//Reset
	IF x_Reset THEN
		x_Speicher:=FALSE;
	END_IF
	
//Ausgang schreiben
	x_Aus:=x_Speicher;

END_FUNCTION_BLOCK

// Converters/Converter2Punkt
(*Der Eingang f_Ein wird anhand des Bereiches von f_Ein_Min f_Ein_Max auf den Bereich f_Aus_Min und f_Aus_Max berechnet und auf den Ausgang f_Aus gegeben.
*)
FUNCTION_BLOCK Converter2Punkt
(*
Versionsverlauf: 
Version		|Autor	|Bemerkung
------------------------------------------------------------------------------------------------------------ 
17.06.00	|ShgB	|erste Freigabe 
17.06.01	|ShgB	|von Integer auf Real geändert 
17.08.00	|LeaF	|Freigabe	

*)
VAR_INPUT
	f_Ein:REAL;//Eingang
	f_Ein_Min:REAL;//Eingangsbereich Minimum
	f_Ein_Max:REAL;//Eingangsbereich Maximum
	f_Aus_Min:REAL;//Ausgangsbereich Minimum
	f_Aus_Max:REAL;//Ausgangsbereich Maximum
END_VAR
VAR_OUTPUT
	f_Aus:REAL;//Ausgang
END_VAR
VAR
END_VAR

IF f_Ein_Max-f_Ein_Min <> 0 THEN
	f_Aus:=(f_Aus_Max-f_Aus_Min)/(f_Ein_Max-f_Ein_Min)*(f_Ein-f_Ein_Min)+f_Aus_Min;
ELSE
	f_Aus:=f_Aus_Max;
END_IF

END_FUNCTION_BLOCK

// Math/Maximum
(*Gibt den grössten der angeschlossenen Werten aus.
*)
FUNCTION_BLOCK Maximum
(*
Versionsverlauf: 
Version		|Autor	|Bemerkung
------------------------------------------------------------------------------------------------------------ 
17.06.00	|Shgb	|erste Freigabe 
17.06.01	|ShgB	|von Integer auf Real geändert	 
17.08.00	|LeaF	|Freigabe

*)
VAR_INPUT
	f_Ein1 :REAL:=0.00001;//Wert 1
	f_Ein2 :REAL:=0.00001;//Wert 2
	f_Ein3 :REAL:=0.00001;//Wert 3
	f_Ein4 :REAL:=0.00001;//Wert 4
	f_Ein5 :REAL:=0.00001;//Wert 5
	f_Ein6 :REAL:=0.00001;//Wert 6
	f_Ein7 :REAL:=0.00001;//Wert 7
	f_Ein8 :REAL:=0.00001;//Wert 8
END_VAR
VAR_OUTPUT
	f_Aus:REAL;//Grösste Wert
END_VAR
VAR
	i_Arraypos:INT;
	af_Array: ARRAY [1..8] OF REAL;
END_VAR

// Werte in Array platzieren
	af_Array[1]:=f_Ein1;
	af_Array[2]:=f_Ein2;
	af_Array[3]:=f_Ein3;
	af_Array[4]:=f_Ein4;
	af_Array[5]:=f_Ein5;
	af_Array[6]:=f_Ein6;
	af_Array[7]:=f_Ein7;
	af_Array[8]:=f_Ein8;
	
//Zahlen die kleiner als 0 sind
	f_Aus := af_Array[1];	
	
//Auswertung der grössten Zahl
	FOR i_Arraypos:=2 TO 8 DO
		IF af_Array[i_Arraypos] >= f_Aus AND af_Array[i_Arraypos] <> 0.00001 THEN
			f_Aus := af_Array[i_Arraypos];
		END_IF
	END_FOR

END_FUNCTION_BLOCK

// Converters/Int_to_Druck
(*Der analoge Wert der Eingangskarte wird von einem 16 bit Integer in einen REAL Wert umgewandelt und ein Offset dazu addiert.
Standardmässig ist der Eingangsbereich von 0 - 32767 eingestellt. Sollte dieser nicht übereinstimmen kann der Bereich angepasst werden.
*)
FUNCTION_BLOCK Int_to_Druck
(*
Versionsverlauf: 
Version		|Autor	|Bemerkung
------------------------------------------------------------------------------------------------------------ 
17.06.00	|Shgb	|erste Freigabe  
17.08.00	|LeaF	|Freigabe

*)
VAR_INPUT
	i_Ein:INT;//Digitaler Eingangswert
END_VAR
VAR_INPUT PERSISTENT
	i_Ein_Min:INT:=0;//Eingangsbereich Minimum
	i_Ein_Max:INT:=32767;//Eingangsbereich Maximum
	f_Aus_Min:REAL;//Minimum des Drucktransmitters
	f_Aus_Max:REAL;//Maximum des Drucktransmitters
	f_Offset:REAL;//Offset der dazu addiert wird
END_VAR
VAR_OUTPUT
	f_Aus:REAL;//Druck im REAL Format
END_VAR
VAR//GUI Variablen
	f_GUI_Input:REAL;
END_VAR

IF i_Ein_Max-i_Ein_Min <> 0 THEN
	f_Aus:=(f_Aus_Max-f_Aus_Min)/(i_Ein_Max-i_Ein_Min)*(i_Ein-i_Ein_Min)+f_Aus_Min+f_Offset;
ELSE
	f_Aus:=f_Aus_Min;
END_IF

f_GUI_Input:=f_Aus-f_Offset;

END_FUNCTION_BLOCK

// Converters/Int_to_Temperature
(*Wandelt die Temperatur im INT Format, die von der Eingangskarte kommt, in eine Temperatur in REAL Format um und rechnet einen Offset dazu.
*)
FUNCTION_BLOCK Int_to_Temperature
(*
Versionsverlauf: 
Version		|Autor	|Bemerkung
------------------------------------------------------------------------------------------------------------ 
17.06.00	|Shgb	|erste Freigabe  
17.08.00	|LeaF	|Freigabe

*)
VAR_INPUT
	i_Ein:INT;//Temperatur von Karte
END_VAR
VAR_INPUT PERSISTENT
	f_Offset:REAL;//Offset der dazu addiert wird
END_VAR
VAR_OUTPUT
	f_Temperatur:REAL;//Ausgang REAL
END_VAR
VAR//GUI Variablen
	f_GUI_Input:REAL;
END_VAR

f_Temperatur:=i_Ein/10.0+f_Offset;
f_GUI_Input:=i_Ein/10.0;

END_FUNCTION_BLOCK

// Converters/Prozent_to_Int
(*Wandelt eine Prozentangabe vom Format REAL in eine Integer Zahl für die analoge Augangskarte um.
Standardmässig ist der Eingangsbereich von 0 - 32767 eingestellt. Sollte dieser nicht übereinstimmen kann der Bereich angepasst werden.
*)
FUNCTION_BLOCK Prozent_to_Int
(*
Versionsverlauf: 
Version		|Autor	|Bemerkung
------------------------------------------------------------------------------------------------------------ 
17.06.00	|Shgb	|erste Freigabe 
17.08.00	|LeaF	|Freigabe 

*)
VAR_INPUT
	f_Ein:REAL;//Eingang in Prozent
END_VAR
VAR_INPUT PERSISTENT
	i_Aus_Min:INT:=0;//Eingangsbereich Minimum
	i_Aus_Max:INT:=32767;//eingangsbereich Maximum
END_VAR
VAR_OUTPUT
	f_Aus:INT;//Ausgang
END_VAR
VAR
END_VAR

f_Aus:=real_to_int((i_Aus_Max-i_Aus_Min)*f_Ein/100.0);

END_FUNCTION_BLOCK

// Converters/Time_to_Timestruct
(*Wandelt die Eingangsvariable vom Typ TIME in ein TIMESTRUCT um.
*)
FUNCTION_BLOCK Time_to_Timestruct
(*
Versionsverlauf: 
Version		|Autor	|Bemerkung
------------------------------------------------------------------------------------------------------------ 
17.06.00	|Shgb	|erste Freigabe 	 
17.08.00	|LeaF	|Freigabe

*)
VAR_INPUT
	t_Ein:TIME;//Eingang
END_VAR
VAR_OUTPUT
	t_Aus:timestruct;//Ausgang
END_VAR
VAR
	OT:OTSTRUCT;
END_VAR

OT:=TIME_TO_OTSTRUCT(t_Ein);
t_Aus.wMilliseconds:=ot.wMilliseconds;
t_Aus.wSecond:=ot.wSecond;
t_Aus.wMinute:=ot.wMinute;
t_Aus.wHour:=ot.wHour;
t_Aus.wDay:=ot.wDay+ot.wWeek*7;

END_FUNCTION_BLOCK

// Converters/Timestruct_to_Time
(*Wandelt einen TIMESTRUCT in die Ausgangsvariable vom Typ TIME um.
*)
FUNCTION_BLOCK Timestruct_to_Time
(*
Versionsverlauf: 
Version		|Autor	|Bemerkung
------------------------------------------------------------------------------------------------------------ 
17.06.00	|Shgb	|erste Freigabe  
17.08.00	|LeaF	|Freigabe	

*)
VAR_INPUT
	t_Ein:timestruct;//Eingang
END_VAR
VAR_OUTPUT
	t_Aus:TIME;//Ausgang
END_VAR
VAR
END_VAR

t_Aus:=DINT_TO_TIME(t_Ein.wMilliseconds
					+ t_Ein.wSecond*1000
					+ t_Ein.wMinute*1000*60
					+ t_Ein.wHour*1000*60*60
					+ t_Ein.wDay*1000*60*60*24);

END_FUNCTION_BLOCK

// Druck_Temp/R1234ze
(*Wandelt den Druck in die Entsprechende Temperatur um. Die Druck-Temperatur Werte sind in der Nassdampftabelle in den Globalen Variablen hinterlegt.
*)
FUNCTION_BLOCK R1234ze
(*
Versionsverlauf: 
Version		|Autor	|Bemerkung
------------------------------------------------------------------------------------------------------------ 
17.06.00	|Shgb	|erste Freigabe 
17.06.01	|ShgB	|von Integer auf Real geändert	 
17.08.00	|LeaF	|Freigabe

*)
VAR_INPUT
	f_ND:REAL;//Druck für Verdampfungstemperatur
	f_HD:REAL;//Druck für Kondensationstemperatur
END_VAR
VAR_OUTPUT
	f_VerdTemp:REAL;//Verdampfungstemperatur
	f_KondTemp:REAL;//Kondensationstemperatur
END_VAR
VAR
END_VAR

//Niederdruck
	f_VerdTemp:=Nassdampftabelle.R1234ze[REAL_TO_INT(f_ND*100)+100]/10.0;
	
//Hochdruck
	f_KondTemp:=Nassdampftabelle.R1234ze[REAL_TO_INT(f_HD*100)+100]/10.0;

END_FUNCTION_BLOCK

// Druck_Temp/R134a
(*Wandelt den Druck in die Entsprechende Temperatur um. Die Druck-Temperatur Werte sind in der Nassdampftabelle in den Globalen Variablen hinterlegt.
*)
FUNCTION_BLOCK R134a
(*
Versionsverlauf: 
Version		|Autor	|Bemerkung
------------------------------------------------------------------------------------------------------------ 
17.06.00	|Shgb	|erste Freigabe 
17.06.01	|ShgB	|von Integer auf Real geändert	 
17.08.00	|LeaF	|Freigabe

*)
VAR_INPUT
	f_ND:REAL;//Druck für Verdampfungstemperatur
	f_HD:REAL;//Druck für Kondensationstemperatur
END_VAR
VAR_OUTPUT
	f_VerdTemp:REAL;//Verdampfungstemperatur
	f_KondTemp:REAL;//Kondensationstemperatur
END_VAR
VAR
END_VAR

//Niederdruck
	f_VerdTemp:=Nassdampftabelle.R134a[REAL_TO_INT(f_ND*100)+100]/10.0;
	
//Hochdruck
	f_KondTemp:=Nassdampftabelle.R134a[REAL_TO_INT(f_HD*100)+100]/10.0;

END_FUNCTION_BLOCK

// Druck_Temp/R407c
(*Wandelt den Druck in die Entsprechende Temperatur um. Die Druck-Temperatur Werte sind in der Nassdampftabelle in den Globalen Variablen hinterlegt.
*)
FUNCTION_BLOCK R407c
(*
Versionsverlauf: 
Version		|Autor	|Bemerkung
------------------------------------------------------------------------------------------------------------ 
17.06.00	|Shgb	|erste Freigabe 
17.06.01	|ShgB	|von Integer auf Real geändert	 
17.08.00	|LeaF	|Freigabe

*)
VAR_INPUT
	f_ND:REAL;//Druck für Verdampfungstemperatur
	f_HD:REAL;//Druck für Kondensationstemperatur
END_VAR
VAR_OUTPUT
	f_VerdTemp:REAL;//Verdampfungstemperatur
	f_KondTemp:REAL;//Kondensationstemperatur
END_VAR
VAR
END_VAR

//Niederdruck
	f_VerdTemp:=Nassdampftabelle.R407cDew[REAL_TO_INT(f_ND*100)+100]/10.0;
	
//Hochdruck
	f_KondTemp:=Nassdampftabelle.R407cBubble[REAL_TO_INT(f_HD*100)+100]/10.0;

END_FUNCTION_BLOCK

// Druck_Temp/R410a
(*Wandelt den Druck in die Entsprechende Temperatur um. Die Druck-Temperatur Werte sind in der Nassdampftabelle in den Globalen Variablen hinterlegt.
*)
FUNCTION_BLOCK R410a
(*
Versionsverlauf: 
Version		|Autor	|Bemerkung
------------------------------------------------------------------------------------------------------------ 
17.06.00	|Shgb	|erste Freigabe 
17.06.01	|ShgB	|von Integer auf Real geändert	 
17.08.00	|LeaF	|Freigabe

*)
VAR_INPUT
	f_ND:REAL;//Druck für Verdampfungstemperatur
	f_HD:REAL;//Druck für Kondensationstemperatur
END_VAR
VAR_OUTPUT
	f_VerdTemp:REAL;//Verdampfungstemperatur
	f_KondTemp:REAL;//Kondensationstemperatur
END_VAR
VAR
END_VAR

//Niederdruck
	f_VerdTemp:=Nassdampftabelle.R410a[REAL_TO_INT(f_ND*100)+100]/10.0;
	
//Hochdruck
	f_KondTemp:=Nassdampftabelle.R410a[REAL_TO_INT(f_HD*100)+100]/10.0;

END_FUNCTION_BLOCK

// Handschaltungen/HS_Bool
(*Handschaltung für BOOL. 0=> Aus, 1=> Ein und 2=> Automatik.
*)
FUNCTION_BLOCK HS_Bool
(*
Versionsverlauf: 
Version		|Autor	|Bemerkung
------------------------------------------------------------------------------------------------------------ 
17.06.00	|Shgb	|erste Freigabe   
17.08.00	|LeaF	|Freigabe

*)
VAR_INPUT
	x_Ein:BOOL;//Eingang
END_VAR
VAR_INPUT PERSISTENT
	i_Modus:INT;//Modusvorgabe
END_VAR
VAR_OUTPUT
	x_Aus:BOOL;//Ausgang
END_VAR
VAR
END_VAR
VAR CONSTANT
	Ein:INT:=1;
	Aus:INT:=0;
	Auto:INT:=2;
END_VAR

CASE i_Modus OF
	Ein:
		x_Aus:=TRUE;
	Aus:
		x_Aus:=FALSE;
	Auto:
		x_Aus:=x_Ein;
ELSE
	x_Aus:=FALSE;
END_CASE;

END_FUNCTION_BLOCK

// Handschaltungen/HS_Int
(*Handschaltung für INT. 1=> Manuell und 2=> Automatik.
*)
FUNCTION_BLOCK HS_Int
(*
Versionsverlauf: 
Version		|Autor	|Bemerkung
------------------------------------------------------------------------------------------------------------ 
17.06.00	|Shgb	|erste Freigabe   
17.08.00	|LeaF	|Freigabe

*)
VAR_INPUT
	i_Ein:INT;//Eingang
END_VAR
VAR_INPUT PERSISTENT
	i_Manu:INT;//Manuelle Sollstellung
	i_Modus:INT;//Modusvorgabe
END_VAR
VAR_OUTPUT
	i_Aus:INT;//Ausgang
END_VAR
VAR
END_VAR
VAR CONSTANT
	Ein:INT:=1;
	Aus:INT:=0;
	Auto:INT:=2;
END_VAR

CASE i_Modus OF
	Ein:
		i_Aus:=i_Manu;
	Auto:
		i_Aus:=i_Ein;
ELSE
	i_Aus:=0;
END_CASE;

END_FUNCTION_BLOCK

// Handschaltungen/HS_Real
(*Handschaltung für REAL. 1=> Manuell und 2=> Automatik.
*)
FUNCTION_BLOCK HS_Real
(*
Versionsverlauf: 
Version		|Autor	|Bemerkung
------------------------------------------------------------------------------------------------------------ 
17.06.00	|Shgb	|erste Freigabe   
17.08.00	|LeaF	|Freigabe

*)
VAR_INPUT
	f_Ein:REAL;//Eingang
END_VAR
VAR_INPUT PERSISTENT
	f_Manu:REAL;//Manuelle Sollstellung
	i_Modus:INT;//Modusvorgabe
END_VAR
VAR_OUTPUT
	f_Aus:real;//Ausgang
END_VAR
VAR
END_VAR
VAR CONSTANT
	Ein:INT:=1;
	Aus:INT:=0;
	Auto:INT:=2;
END_VAR

CASE i_Modus OF
	Ein:
		f_Aus:=f_Manu;
	Auto:
		f_Aus:=f_Ein;
ELSE
	f_Aus:=0;
END_CASE;

END_FUNCTION_BLOCK

// Heizen_Kuehlen/FG_Heizen
(* Mit der Tagesschaltuhr wird der Tag_Nacht Sollwert bestimmt. Schaltuhr Ein = Nachtbetrieb. Der Funktionsblock wird mit dem Eingang x_Akt aktiviert.
 Unterschreitet die Aussentemperatur und die gemittelte AT den einstellbaren Sollwert
 in der fix eingestellten Zeit von 5 Minuten, schaltet der Einschaltbefehl bis die beiden Temperatur Werte
 der eingestellten Sollwert wieder überschreiten. 
 *)
FUNCTION_BLOCK FG_Heizen
(*
Versionsverlauf: 
Version		|Autor	|Bemerkung
------------------------------------------------------------------------------------------------------------ 
17.07.00	|KuzR	|erste Freigabe  
17.08.00	|LeaF	|Freigabe

*)
VAR_INPUT 
	x_Nacht:BOOL;//Ein=Nacht, Aus=Tag
	f_AT:REAL;//Aussentemperatur
	f_RT_AT:REAL;//Berechnete Aussentemperatur
END_VAR
VAR_INPUT PERSISTENT
	x_Akt_FB:BOOL := TRUE;//Aktivierung FB
	f_SW_Tag:REAL := 20;//Sollwert Tag
	f_SW_Nacht:REAL := 16;//Sollwert Nacht
END_VAR
VAR_OUTPUT
	x_EB:BOOL;//Einschaltbefehl
END_VAR
VAR
	f_Aus_SW_Tag_Nacht:REAL;
	x_EIN_Timer:BOOL;
	Timer:TON;
	MUX_B: MUX_B;
	CLK_D: CLK_D;
	Timestruct_to_Time: Timestruct_to_Time;
	t_time: TIME;
	x_FG_Tag:BOOL;
	x_FG_Nacht:BOOL;
END_VAR

//Nachtakivierung
	x_FG_Nacht:=x_Akt_FB AND x_Nacht;
	
//Tagaktivierung	
	x_FG_Tag:=x_Akt_FB AND NOT x_Nacht;
	
//Tag/Nacht Umschaltung
	MUX_B(
	f_Ein_1:=f_SW_Tag , 
	f_Ein_2:=f_SW_Nacht , 
	x_Ein_1:=x_FG_Tag , 
	x_Ein_2:=x_FG_Nacht , 
	f_Aus=>f_Aus_SW_Tag_Nacht );	

//Temperaturen Abfrage Tag_Nacht und Timer einschalten
	x_EIN_Timer:= x_Akt_FB AND  f_AT < f_Aus_SW_Tag_Nacht AND f_RT_AT < f_Aus_SW_Tag_Nacht;
		
//Timer Restzeit für Abfrage AT und SW
	Timer(in:=x_EIN_Timer , pt:=T#5M);	

//Einschaltbefehl 	
	x_EB:=Timer.Q;

END_FUNCTION_BLOCK

// Uhren/CLK_D
(*Uhr mit Tagesprogramm. Einschaltzeit => t_Ein.wHour, t_ein.wMinute und Ausschaltzeit => t_Aus.wHour und t_Aus.wMinute. Eingabe im Timestruct Format.
Vergleicht Ein- und Ausschaltzeit mit der Globalen_Uhr(Globale Variable)
*)
FUNCTION_BLOCK CLK_D
(*
Versionsverlauf: 
Version		|Autor	|Bemerkung
------------------------------------------------------------------------------------------------------------ 
17.06.00	|KuzR	|erste Freigabe 
17.08.00	|LeaF	|Freigabe

*)
VAR_INPUT Persistent
	t_Ein:timestruct;//Eingabe Einschaltzeit 
	t_Aus:timestruct;//Eingabe Ausschaltzeit 
END_VAR
VAR_OUTPUT
	x_Aus:BOOL;//Digitaler Ausgang		 
END_VAR
VAR
END_VAR

//schaltet jeden Tag ein, eingestell e Zeit  
	IF Globale_Uhr.systemtimestruct.wHour = t_Ein.wHour AND
 	   Globale_Uhr.systemtimestruct.wMinute >= t_Ein.wMinute THEN
			x_Aus:= TRUE;
	END_IF
				
//schaltet jeden Tag wieder aus, eingestellte Zeit			
	IF 	Globale_Uhr.systemtimestruct.wHour = t_Aus.wHour AND
		Globale_Uhr.systemtimestruct.wMinute >= t_Aus.wMinute THEN
			x_Aus:= FALSE;
	END_IF

END_FUNCTION_BLOCK

// Heizen_Kuehlen/FG_Kuehlen
(* Mit der Tagesschaltuhr wird der Tag_Nacht Sollwert bestimmt. Schaltuhr Ein = Nachtbetrieb. Der Funktionsblock wird mit dem Eingang x_Akt aktiviert.
 Überschreitet die Aussentemperatur und die gemittelte AT den einstellbaren Sollwert
 in der fix eingestellten Zeit von 5 Min und der Eingang x_Absch_Hz_Kue war länger nicht angezogen, schaltet der Einschaltbefehl bis die beiden Temperatur Werte
 der eingestellten Sollwert wieder unterschreiten. 
 *)
FUNCTION_BLOCK FG_Kuehlen
(*
Versionsverlauf: 
Version		|Autor	|Bemerkung
------------------------------------------------------------------------------------------------------------ 
17.07.00	|KuzR	|erste Freigabe  
17.08.00	|LeaF	|Freigabe

*)
VAR_INPUT 
	f_AT:REAL;//Aussentemperatur
	f_RT_AT:REAL;//Berechnete Aussentemperatur
END_VAR
VAR_INPUT PERSISTENT
	x_Akt_FB:BOOL := true;//Aktivierung FB
	x_Nacht: BOOL;//Ein=Nacht, Aus=Tag
	f_SW_Tag:REAL := 10;//Sollwert Tag
	f_SW_Nacht:REAL := 10;//Sollwert Nacht
	x_Absch_HZ_Kue:BOOL;//Abschaltung HZ und Kühlen
END_VAR
VAR_OUTPUT
	x_EB:BOOL;//Einschaltbefehl
END_VAR
VAR
	f_Aus_SW_Tag_Nacht:REAL;
	x_Tag_Nacht:BOOL;
	x_EIN_Timer:BOOL;
	Timer:TON;
	MUX_B: MUX_B;
	CLK_D: CLK_D;
	Timestruct_to_Time: Timestruct_to_Time;
	t_time: TIME;
	x_FG_Tag:BOOL;//Freigabe Tag
	x_FG_Nacht:BOOL;//Freigabe Nacht
END_VAR

//Nachtakivierung
	x_FG_Nacht:=x_Akt_FB AND x_Nacht;
	
//Tagaktivierung	
	x_FG_Tag:=x_Akt_FB AND NOT x_Nacht;
	
//Tag/Nacht Umschaltung
	MUX_B(
	f_Ein_1:=f_SW_Tag , 
	f_Ein_2:=f_SW_Nacht , 
	x_Ein_1:=x_FG_Tag , 
	x_Ein_2:=x_FG_Nacht , 
	f_Aus=>f_Aus_SW_Tag_Nacht );	

//Temperaturen Abfrage Tag_Nacht und Timer einschalten
	x_EIN_Timer:= x_Akt_FB AND  f_AT > f_Aus_SW_Tag_Nacht AND f_RT_AT > f_Aus_SW_Tag_Nacht AND NOT x_Absch_HZ_Kue;
		
//Timer Restzeit für Abfrage AT und SW
	Timer(in:=x_EIN_Timer , pt:=T#5M);	

//Einschaltbefehl 	
	x_EB:=Timer.Q;

END_FUNCTION_BLOCK

// Heizen_Kuehlen/GR_2
//Kühlkurve, mit 2 AT-Punkten wird ein Tag, bzw. Nachtsollwert berechnet. Referenpunkt T01 muss grösser sein Als T02
//Umschaltbar Tag/Nacht Aktivierung. Sollwert Max und Min Begrenzung. 
FUNCTION_BLOCK GR_2
(*
Versionsverlauf: 
Version		|Autor	|Bemerkung
------------------------------------------------------------------------------------------------------------ 
17.06.00	|KuzR	|erste Freigabe  
17.08.00	|LeaF	|Freigabe

*)
VAR_INPUT
	f_AT:REAL;//Aussentempertur
	x_Akt_Nacht:BOOL;//Nachtakivierung	
END_VAR
VAR_INPUT PERSISTENT
	f_RefPunkt_TO1:REAL;//Referenzpunkt T01 AT
	f_SW_W1_Tag:REAL;//Sollwertpunkt 1 Tag
	f_SW_W1_Nacht:REAL;//Sollwertpunkt 1 Nacht
	f_RefPunkt_TO2:REAL;//Referenzpunkt T02 AT
	f_SW_W2_Tag:REAL;//Sollwertpunkt 2 Tag
	f_SW_W2_Nacht:REAL;//Sollwertpunkt 1 Nacht
	f_SW_Max:REAL;//Sollwert Max.
	f_SW_Min:REAL;//Sollwert Min.
END_VAR
VAR_OUTPUT
	f_SW_Ber:REAL;//Ausgang Sollwert
END_VAR
	
VAR
	
	Converter2Punkt: Converter2Punkt;
END_VAR

//T01 muss Höher sein als T02
//Aussentemperatur T2-T1, Tag
//Aussentemperatur < T1 oder Aussentemperatur > T2 für Min/Max Begrenzung
	IF NOT x_Akt_Nacht AND  f_RefPunkt_TO2 <= f_AT AND f_RefPunkt_TO1 > f_AT OR NOT x_Akt_Nacht AND f_AT < f_RefPunkt_TO1 OR NOT x_Akt_Nacht AND f_AT > f_RefPunkt_TO2  THEN 
		Converter2Punkt(
	f_Ein:=f_AT , 
	f_Ein_Min:=f_RefPunkt_TO1 , 
	f_Ein_Max:=f_RefPunkt_TO2 , 
	f_Aus_Min:=f_SW_W1_Tag , 
	f_Aus_Max:=f_SW_W2_Tag , 
	f_Aus=>f_SW_Ber );
	END_IF
	
//Aussentemperatur T2-T1, Nacht
//Aussentemperatur < T1 oder Aussentemperatur > T2 für Min/Max Begrenzung
	IF  x_Akt_Nacht AND  
		f_RefPunkt_TO2 <= f_AT AND 
		f_RefPunkt_TO1 > f_AT OR  x_Akt_Nacht AND f_AT < f_RefPunkt_TO1 OR x_Akt_Nacht AND f_AT < f_RefPunkt_TO1 OR  x_Akt_Nacht AND f_AT > f_RefPunkt_TO2  THEN 
		Converter2Punkt(
	f_Ein:=f_AT , 
	f_Ein_Min:=f_RefPunkt_TO1 , 
	f_Ein_Max:=f_RefPunkt_TO2 , 
	f_Aus_Min:=f_SW_W1_Nacht , 
	f_Aus_Max:=f_SW_W2_Nacht , 
	f_Aus=>f_SW_Ber );
	END_IF
	
//Min/Max Begrenzung 
	f_SW_Ber := LIMIT(f_SW_Min,f_SW_Ber, f_SW_Max);

END_FUNCTION_BLOCK

// Heizen_Kuehlen/GR_4_mit_RE
(* Heizkurve mit Raumeinfluss vergleicht Aussentemperatur zwischen den Sollwerten. Referenzpunkt T01 muss die kleinste Temperatur-,bzw. T04 die grösste Temperatur sein.
 Anhand von vier AT Punkten wird der Tag-, bzw. Nachtsollwert berechnet.
 Umschaltbar Tag/Nacht Aktivierung. Sollwert mit  Max und Min Begrenzung. Maximale negative Korrektur (i_MaxKorrNeg) muss zwingend als negativen Wert eingegeben werden und Maximale positive  Korrektur als positiven Wert.
*)
FUNCTION_BLOCK GR_4_mit_RE
(*
Versionsverlauf: 
Version		|Autor	|Bemerkung
------------------------------------------------------------------------------------------------------------ 
17.06.00	|KuzR	|erste Freigabe  
17.08.00	|LeaF	|Freigabe

*)
VAR_INPUT
	f_AT:REAL; //Aussentemperatur
	x_Akt_Nacht:BOOL;	// Nachtakivierung
	f_MT_Raum:REAL; // Raumtemperatur
END_VAR
VAR_INPUT PERSISTENT	
	f_RefPunkt_TO1:REAL; // Referenzpunkt T01 AT
	f_SW_W1_Tag:REAL; // Sollwertpunkt 1 Tag
	f_SW_W1_Nacht:REAL; // Sollwertpunkt 1 Nacht
	f_RefPunkt_TO2:REAL; // Referenzpunkt T02 AT
	f_SW_W2_Tag:REAL; // Sollwertpunkt 2 Tag
	f_SW_W2_Nacht:REAL; // Sollwertpunkt 2 Nacht
	f_RefPunkt_TO3:REAL; // Referenzpunkt T03 AT
	f_SW_W3_Tag:REAL; // Sollwertpunkt 3 Tag
	f_SW_W3_Nacht:REAL; // Sollwertpunkt 3 Nacht
	f_RefPunkt_TO4:REAL; // Referenzpunkt T04 AT
	f_SW_W4_Tag:REAL; // Sollwertpunkt 4 Tag
	f_SW_W4_Nacht:REAL; // Sollwertpunkt 4 Nacht
	f_SW_Max:REAL; // Sollwert Max.
	f_SW_Min:REAL; //Sollwert Min.
	f_KorrFaktor:REAL;  // Korrekturfaktor
	i_MaxKorrPos:INT; // Max. Pos. Korrektur(muss positiver Wert sein)
	i_MaxKorrNeg:INT; // Max. Neg. Korrektur(muss negativer Wert sein)
	f_SW_Raum:REAL;	// Sollwert Raum
END_VAR
VAR_OUTPUT
	f_SW_Ber:REAL; // Sollwert Berechnung
	f_SW_Korr:REAL; // Korrigierte Sollwertberechnung
END_VAR
VAR
	f_Diff:REAL;
	f_Diff_faktor:REAL;
	Converter2Punkt: Converter2Punkt;
END_VAR

//Aussentemperatur T4-T3, Tag
//Aussentemperatur > T4, für Max Sollwert Berechnung
	IF NOT x_Akt_Nacht AND f_RefPunkt_TO4 > f_AT AND f_RefPunkt_TO3 <= f_AT OR NOT x_Akt_Nacht AND f_AT >= f_RefPunkt_TO4 THEN
		Converter2Punkt( 
	f_Ein:=f_AT , 
	f_Ein_Min:=f_RefPunkt_TO3 , 
	f_Ein_Max:=f_RefPunkt_TO4 , 
	f_Aus_Min:=f_SW_W3_Tag , 
	f_Aus_Max:=f_SW_W4_Tag , 
	f_Aus=>f_SW_Ber );
	END_IF
//Aussentemperatur T4-T3, Nacht
//Aussentemperatur > T4, für Max Sollwert Berechnung
	IF x_Akt_Nacht AND f_RefPunkt_TO4 > f_AT AND f_RefPunkt_TO3 <= f_AT OR x_Akt_Nacht AND f_AT >= f_RefPunkt_TO4 THEN
		Converter2Punkt(
	f_Ein:=f_AT , 
	f_Ein_Min:=f_RefPunkt_TO3 , 
	f_Ein_Max:=f_RefPunkt_TO4 , 
	f_Aus_Min:=f_SW_W3_Nacht , 
	f_Aus_Max:=f_SW_W4_Nacht , 
	f_Aus=>f_SW_Ber );
	END_IF
//Aussentemperatur T3-T2, Tag
	IF NOT x_Akt_Nacht AND  f_RefPunkt_TO3 > f_AT AND f_RefPunkt_TO2 <= f_AT THEN
		Converter2Punkt(
	f_Ein:=f_AT , 
	f_Ein_Min:=f_RefPunkt_TO2 , 
	f_Ein_Max:=f_RefPunkt_TO3 , 
	f_Aus_Min:=f_SW_W2_Tag , 
	f_Aus_Max:=f_SW_W3_Tag , 
	f_Aus=>f_SW_Ber );
	END_IF
//Aussentemperatur T3-T2, Nacht
	IF x_Akt_Nacht AND  f_RefPunkt_TO3 > f_AT AND f_RefPunkt_TO2 <= f_AT THEN
		Converter2Punkt(
	f_Ein:=f_AT , 
	f_Ein_Min:=f_RefPunkt_TO2 , 
	f_Ein_Max:=f_RefPunkt_TO3 , 
	f_Aus_Min:=f_SW_W2_Nacht , 
	f_Aus_Max:=f_SW_W3_Nacht , 
	f_Aus=>f_SW_Ber );
	END_IF	
//Aussentemperatur T2-T1, Tag
//Aussentemperatur < T1, für Min Sollwert Berechnung
	IF NOT x_Akt_Nacht AND f_RefPunkt_TO2 > f_AT AND f_RefPunkt_TO1 <= f_AT OR NOT x_Akt_Nacht AND f_AT < f_RefPunkt_TO1  THEN
		Converter2Punkt(
	f_Ein:=f_AT , 
	f_Ein_Min:=f_RefPunkt_TO1 , 
	f_Ein_Max:=f_RefPunkt_TO2 , 
	f_Aus_Min:=f_SW_W1_Tag , 
	f_Aus_Max:=f_SW_W2_Tag , 
	f_Aus=>f_SW_Ber );
	END_IF
//Aussentemperatur T2-T1, Nacht
//Aussentemperatur < T1, für Min Sollwert Berechnung
	IF x_Akt_Nacht AND f_RefPunkt_TO2 > f_AT AND f_RefPunkt_TO1 <= f_AT OR x_Akt_Nacht AND f_AT < f_RefPunkt_TO1  THEN
		Converter2Punkt(
	f_Ein:=f_AT , 
	f_Ein_Min:=f_RefPunkt_TO1 , 
	f_Ein_Max:=f_RefPunkt_TO2 , 
	f_Aus_Min:=f_SW_W1_Nacht , 
	f_Aus_Max:=f_SW_W2_Nacht , 
	f_Aus=>f_SW_Ber );
	END_IF

//Korrektur Raumtemperatur
	f_Diff:= f_SW_Raum-f_MT_Raum;
	
//Maximale_Minimale Korrektur
	IF f_Diff > i_MaxKorrPos THEN
		f_Diff:=i_MaxKorrPos;
	END_IF
	IF f_Diff < i_MaxKorrNeg THEN
		f_Diff:=i_MaxKorrNeg;
	END_IF
	
	f_Diff_faktor:=f_Diff*f_KorrFaktor;
	
//Begrenzung für positive und negative Begerenzung
	IF f_Diff_faktor > i_MaxKorrPos THEN
		f_Diff_faktor:=i_MaxKorrPos;
	END_IF
	IF f_Diff_faktor < i_MaxKorrNeg THEN
		f_Diff_faktor:=i_MaxKorrNeg;
	END_IF
	
//Korrrigierter Sollwert	
	f_SW_Korr:=f_SW_Ber + f_Diff_faktor ;

//Max Begrenzung 	
	IF f_SW_Korr >= f_SW_Max THEN
		f_SW_Korr:=f_SW_Max; 
	END_IF	
//Min Begrenzung 
	IF f_SW_Korr < f_SW_Min THEN
		f_SW_Korr:=f_SW_Min;
	END_IF

END_FUNCTION_BLOCK

// Heizen_Kuehlen/GR_4_ohne_RE
(* Heizkurve ohne Raumeinfluss vergleicht Aussentemperatur zwischen den Sollwerten. Referenzpunkt T01 muss die kleinste Temperatur-,bzw. T04 die grösste Temperatur sein.
 Anhand von vier AT Punkten wird der Tag-, bzw. Nachtsollwert berechnet.
 Umschaltbar Tag/Nacht Aktivierung. Sollwert MAX und MIN Begrenzung.
*)
FUNCTION_BLOCK GR_4_ohne_RE
(*
Versionsverlauf: 
Version		|Autor	|Bemerkung
------------------------------------------------------------------------------------------------------------ 
17.06.00	|KuzR	|erste Freigabe  
17.08.00	|LeaF	|Freigabe

*)
VAR_INPUT
	f_AT:REAL; //Aussentemperatur
	x_Akt_Nacht:BOOL;//Nachtakivierung
END_VAR
VAR_INPUT PERSISTENT
	f_RefPunkt_TO1:REAL;//Referenzpunkt T01 AT
	f_SW_W1_Tag:REAL;//Sollwertpunkt 1 Tag
	f_SW_W1_Nacht:REAL;//Sollwertpunkt 1 Nacht
	f_RefPunkt_TO2:REAL;//Referenzpunkt T02 AT
	f_SW_W2_Tag:REAL;//Sollwertpunkt 2 Tag
	f_SW_W2_Nacht:REAL;//Sollwertpunkt 2 Nacht
	f_RefPunkt_TO3:REAL;//Referenzpunkt T03 AT
	f_SW_W3_Tag:REAL;//Sollwertpunkt 3 Tag
	f_SW_W3_Nacht:REAL;//Sollwertpunkt 3 Nacht
	f_RefPunkt_TO4:REAL;//Referenzpunkt T04 AT
	f_SW_W4_Tag:REAL;//Sollwertpunkt 4 Tag
	f_SW_W4_Nacht:REAL;//Sollwertpunkt 4 Nacht
	f_SW_Max:REAL;//Sollwert Max.
	f_SW_Min:REAL;//Sollwert Min.
END_VAR
VAR_OUTPUT
	f_SW_Ber:REAL;//Sollwert Berechnung
END_VAR
VAR
	Converter2Punkt: Converter2Punkt;
END_VAR

//Aussentemperatur T4-T3, Tag
//Aussentemperatur > T4, für Max Sollwert Berechnung
	IF NOT x_Akt_Nacht AND f_RefPunkt_TO4 > f_AT AND f_RefPunkt_TO3 <= f_AT OR NOT x_Akt_Nacht AND f_AT >= f_RefPunkt_TO4 THEN
		Converter2Punkt( 
	f_Ein:=f_AT , 
	f_Ein_Min:=f_RefPunkt_TO3 , 
	f_Ein_Max:=f_RefPunkt_TO4 , 
	f_Aus_Min:=f_SW_W3_Tag , 
	f_Aus_Max:=f_SW_W4_Tag , 
	f_Aus=>f_SW_Ber );
	END_IF
//Aussentemperatur T4-T3, Nacht
//Aussentemperatur > T4, für Max Sollwert Berechnung
	IF x_Akt_Nacht AND f_RefPunkt_TO4 > f_AT AND f_RefPunkt_TO3 <= f_AT OR x_Akt_Nacht AND f_AT >= f_RefPunkt_TO4 THEN
		Converter2Punkt(
	f_Ein:=f_AT , 
	f_Ein_Min:=f_RefPunkt_TO3 , 
	f_Ein_Max:=f_RefPunkt_TO4 , 
	f_Aus_Min:=f_SW_W3_Nacht , 
	f_Aus_Max:=f_SW_W4_Nacht , 
	f_Aus=>f_SW_Ber );
	END_IF
//Aussentemperatur T3-T2, Tag
	IF NOT x_Akt_Nacht AND  f_RefPunkt_TO3 > f_AT AND f_RefPunkt_TO2 <= f_AT THEN
		Converter2Punkt(
	f_Ein:=f_AT , 
	f_Ein_Min:=f_RefPunkt_TO2 , 
	f_Ein_Max:=f_RefPunkt_TO3 , 
	f_Aus_Min:=f_SW_W2_Tag , 
	f_Aus_Max:=f_SW_W3_Tag , 
	f_Aus=>f_SW_Ber );
	END_IF
//Aussentemperatur T3-T2, Nacht
	IF x_Akt_Nacht AND  f_RefPunkt_TO3 > f_AT AND f_RefPunkt_TO2 <= f_AT THEN
		Converter2Punkt(
	f_Ein:=f_AT , 
	f_Ein_Min:=f_RefPunkt_TO2 , 
	f_Ein_Max:=f_RefPunkt_TO3 , 
	f_Aus_Min:=f_SW_W2_Nacht , 
	f_Aus_Max:=f_SW_W3_Nacht , 
	f_Aus=>f_SW_Ber );
	END_IF	
//Aussentemperatur T2-T1, Tag
//Aussentemperatur < T1, für Min Sollwert Berechnung
	IF NOT x_Akt_Nacht AND f_RefPunkt_TO2 > f_AT AND f_RefPunkt_TO1 <= f_AT OR NOT x_Akt_Nacht AND f_AT < f_RefPunkt_TO1  THEN
		Converter2Punkt(
	f_Ein:=f_AT , 
	f_Ein_Min:=f_RefPunkt_TO1 , 
	f_Ein_Max:=f_RefPunkt_TO2 , 
	f_Aus_Min:=f_SW_W1_Tag , 
	f_Aus_Max:=f_SW_W2_Tag , 
	f_Aus=>f_SW_Ber );
	END_IF
//Aussentemperatur T2-T1, Nacht
//Aussentemperatur < T1, für Min Sollwert Berechnung
	IF x_Akt_Nacht AND f_RefPunkt_TO2 > f_AT AND f_RefPunkt_TO1 <= f_AT OR x_Akt_Nacht AND f_AT < f_RefPunkt_TO1  THEN
		Converter2Punkt(
	f_Ein:=f_AT , 
	f_Ein_Min:=f_RefPunkt_TO1 , 
	f_Ein_Max:=f_RefPunkt_TO2 , 
	f_Aus_Min:=f_SW_W1_Nacht , 
	f_Aus_Max:=f_SW_W2_Nacht , 
	f_Aus=>f_SW_Ber );
	END_IF

//Min/Max Begrenzung 	
	f_SW_Ber := LIMIT(f_SW_Min,f_SW_Ber, f_SW_Max);

END_FUNCTION_BLOCK

// Heizen_Kuehlen/REG2_HEIZEN
(*2 Punkt Regler Heizen
Für Direkt, x_Akt auf true, schaltet der Ausgang auf true. Ist der eingegebene Sollwert addiert mit dem Einschaltpunkt(zB -2) grösser oder gleich der Messtemperatur,
schaltet der digitale Ausgang auf true. Ist der Sollwert addiert mit dem Ausschaltpunkt kleiner oder gleich dem Messwert, schaltet der digitale Ausganf auf false.
*)
FUNCTION_BLOCK REG2_HEIZEN
(*
Versionsverlauf: 
Version		|Autor	|Bemerkung
------------------------------------------------------------------------------------------------------------ 
17.06.00	|KuzR	|erste Freigabe  
17.08.00	|LeaF	|Freigabe

*)
VAR_INPUT
	f_MT:REAL;//Eingang Messwert
END_VAR
VAR_INPUT PERSISTENT
	f_SW:REAL;//Eingang Sollwert
	f_Einschaltpunkt:REAL;//Eingang Einschaltpunkt
	f_Ausschaltpunkt:REAL;//Eingang Ausschaltpunkt
	x_Akt:BOOL;//Direkt-Indirekt Aktivierung
END_VAR
VAR_OUTPUT
	x_Aus:BOOL;//Digitaler Ausgang
END_VAR
VAR
END_VAR

//Direkt- Indirekt Schaltung
	IF   NOT x_Akt THEN 
		x_Aus:=FALSE;
//Einschalten
	ELSIF  f_MT <= f_SW + f_Einschaltpunkt THEN
		x_Aus:= TRUE;
//Ausschalten	
	ELSIF	f_MT  >= f_SW + f_Ausschaltpunkt THEN
		x_Aus:= FALSE;
	END_IF

END_FUNCTION_BLOCK

// Heizen_Kuehlen/REG2_KUEHLEN
(*2 Punkt Regler Kühlen
Für Direkt, x_Akt auf true, schaltet der Ausgang auf true. Ist der eingegebene Sollwert addiert mit dem Einschaltpunkt(zB -2) kleiner oder gleich der Messtemperatur,
schaltet der digitale Ausgang auf true. Ist der Sollwert addiert mit dem Ausschaltpunkt grösser oder gleich dem Messwert, schaltet der digitale Ausganf auf false.
*)
FUNCTION_BLOCK REG2_KUEHLEN
(*
Versionsverlauf: 
Version		|Autor	|Bemerkung
------------------------------------------------------------------------------------------------------------ 
17.06.00	|KuzR	|erste Freigabe  
17.08.00	|LeaF	|Freigabe

*)
VAR_INPUT
	f_MT:REAL;//Eingang Messwert
END_VAR
VAR_INPUT PERSISTENT
	f_SW:REAL;//Eingang Sollwert
	f_Einschaltpunkt:REAL;//Eingang Einschaltpunkt
	f_Ausschaltpunkt:REAL;//Eingang Ausschaltpunkt
	x_Akt:BOOL;//Direkt-Indirekt Aktivierung
END_VAR
VAR_OUTPUT
	x_Aus:BOOL;//Digitaler Ausgang
END_VAR
VAR
END_VAR

//Direkt- Indirekt Schaltung
	IF   NOT x_Akt THEN 
		x_Aus:=FALSE;	
//Einschalten
	ELSIF  f_MT >= f_SW + f_Einschaltpunkt THEN
		x_Aus:= TRUE;	
//Ausschalten	
	ELSIF	f_MT  <= f_SW + f_Ausschaltpunkt THEN
		x_Aus:= FALSE;	
	END_IF

END_FUNCTION_BLOCK

// Heizen_Kuehlen/RT_AT_48
(*Berechnet die gemittelte Aussentemperatur. Die Datensätze für die Mittelwertberechnung ist auf 48 Datensätze ausgelegt.
x_start für die Initialisierung der Aussentemperatur. Mit t_time kann die Zeit bestimmt werden, wann einen Wert ins Array geschrieben werden kann.
*)
FUNCTION_BLOCK RT_AT_48
(*
Versionsverlauf: 
Version		|Autor	|Bemerkung
------------------------------------------------------------------------------------------------------------ 
17.07.00	|KuzR	|erste Freigabe  
17.08.00	|LeaF	|Freigabe

*)
VAR_INPUT
	x_start: BOOL;//Start für die  Initialisierung
	f_AT:REAL;//Eingang Aussentemperatur
END_VAR
VAR_INPUT PERSISTENT	
	t_time:timestruct;//Zeiteingabe 1h oder 24h
END_VAR
VAR_OUTPUT
	f_AT_RT: REAL;//Ausgang gemittelt
END_VAR
VAR 
	i_Ind: INT;
	f_Summe:REAL;
	timer:ton;
	daten:ARRAY [1..i_Datensaetze] OF REAL;
	Timestruct_to_Time:Timestruct_to_Time;	
	x_Flanke: BOOL;
END_VAR
VAR CONSTANT
	i_Datensaetze:INT:=48;
END_VAR

//Für Aussentemperatur Initialisierung muss x_start gedrückt werden
	 IF x_start  THEN
//Grösse des Array für den Mittelwert bestimmen
		 FOR i_Ind:= 1 TO I_DATENSAETZE DO
			 daten[i_Ind]:= f_AT;
		 END_FOR
	 END_IF
	x_start:=FALSE;
//Timestruct to Time
	timestruct_to_time(t_Ein:=t_time);
//Timer läuft immer
	Timer(IN := NOT Timer.Q, PT :=timestruct_to_time.t_Aus/48 );

	IF Timer.Q THEN
    f_Summe := 0;
//die neuen Temperaturwerte werden ins Array geschrieben
    FOR i_Ind := I_DATENSAETZE TO 2 BY -1  DO
        Daten[i_Ind] := Daten[i_Ind - 1];
        f_Summe := f_Summe + Daten[i_Ind];
    END_FOR
//Rechentemperatur berechnen
    Daten[1] := f_AT;
    f_Summe := f_Summe + f_AT;
    f_AT_RT:=f_summe / I_DATENSAETZE;
	END_IF

END_FUNCTION_BLOCK

// Initialisierung/Globale_Zeit
FUNCTION_BLOCK Globale_Zeit
(*
Versionsverlauf: 
Version		|Autor	|Bemerkung
------------------------------------------------------------------------------------------------------------ 
17.06.00	|KuzR	|erste Freigabe 
17.06.01	|ShgB	|Date and Time ergänzt 
17.08.00	|LeaF	|Freigabe

*)
VAR_INPUT Persistent
	tzi_ZeitZone:ST_TimeZoneInformation :=WEST_EUROPE_TZI;
END_VAR
VAR_OUTPUT		 
END_VAR
VAR
	  fbgetSystemTime:getsystemtime;
  	  fileTime:T_FILETIME;
	  
      eTzID:E_TimeZoneID := eTimeZoneID_Unknown;
      fbToLocal:FB_FileTimeToTzSpecificLocalTime;
	  tzInfo:ST_TimeZoneInformation;
END_VAR

//CPU Zeit
	fbgetSystemTime	(timeLoDW=>fileTime.dwLowDateTime, timeHiDW=>fileTime.dwHighDateTime );
	
//Zeitumrechnung
	fbToLocal( in := filetime , tzInfo := tzi_ZeitZone );
	
//Globale Variable, Aktuelle Uhrzeit
	Globale_Uhr.systemtimestruct := FILETIME_TO_systemtime( fbToLocal.out  );
	Globale_Uhr.systemDateAndTime:= FILETIME_TO_DT(fbToLocal.out);

END_FUNCTION_BLOCK

// Math/Average
(*Gibt den Durchschnitt der angeschlossenen Werten aus.
*)
FUNCTION_BLOCK Average
(*
Versionsverlauf: 
Version		|Autor	|Bemerkung
------------------------------------------------------------------------------------------------------------ 
17.06.00	|Shgb	|erste Freigabe  
17.08.00	|LeaF	|Freigabe

*)
VAR_INPUT
	f_Ein1 :REAL:=0.00001;//Wert 1
	f_Ein2 :REAL:=0.00001;//Wert 2
	f_Ein3 :REAL:=0.00001;//Wert 3
	f_Ein4 :REAL:=0.00001;//Wert 4
	f_Ein5 :REAL:=0.00001;//Wert 5
	f_Ein6 :REAL:=0.00001;//Wert 6
	f_Ein7 :REAL:=0.00001;//Wert 7
	f_Ein8 :REAL:=0.00001;//Wert 8
END_VAR
VAR_OUTPUT
	f_Aus:REAL;//Durchschnitt
END_VAR
VAR
	i_Arraypos:INT;
	af_Array: ARRAY [1..8] OF REAL;
	COUNT: COUNT;
END_VAR

// Werte in Array platzieren
	af_Array[1]:=f_Ein1;
	af_Array[2]:=f_Ein2;
	af_Array[3]:=f_Ein3;
	af_Array[4]:=f_Ein4;
	af_Array[5]:=f_Ein5;
	af_Array[6]:=f_Ein6;
	af_Array[7]:=f_Ein7;
	af_Array[8]:=f_Ein8;
	
//Zurücksetzen
	f_Aus:=0;
	
//Anzahl Eingänge zählen
	COUNT(
	x_Ein_1:= f_Ein1<>0.00001, //0.00001 bedeutet nicht aktiv
	x_Ein_2:= f_Ein2<>0.00001, 
	x_Ein_3:= f_Ein3<>0.00001, 
	x_Ein_4:= f_Ein4<>0.00001, 
	x_Ein_5:= f_Ein5<>0.00001, 
	x_Ein_6:= f_Ein6<>0.00001, 
	x_Ein_7:= f_Ein7<>0.00001, 
	x_Ein_8:= f_Ein8<>0.00001);
	
//Summe bilden
	FOR i_Arraypos:=1 TO count.i_Aus DO
		f_Aus:=f_Aus+af_Array[i_Arraypos];
	END_FOR
	
//Durchschnitt berechnen
	IF count.i_Aus >0 THEN
		f_Aus:=f_Aus/count.i_Aus;
	END_IF

END_FUNCTION_BLOCK

// Math/Filter
(*Berechnet die gefilterte Aussentemperatur. x_start für die Initialisierung der Aussentemperatur. Mit t_time kann die Zeit bestimmt werden, wann einen Wert ins Array geschrieben werden kann.
*)
FUNCTION_BLOCK Filter
(*
Versionsverlauf:
Version		|Autor	|Bemerkung
------------------------------------------------------------------------------------------------------------ 
17.07.00	|KuzR	|erste Freigabe  
17.08.00	|LeaF	|Freigabe

*)
VAR_INPUT
	x_start: BOOL;//Start für die  Initialisierung
	f_AT:REAL;//Eingang Aussentemperatur
END_VAR
VAR_INPUT PERSISTENT	
	t_time:timestruct := (wHour := 1);//Takt, wenn ein AT Wert geschrieben wird
END_VAR
VAR_OUTPUT
	f_Aus: REAL;//Ausgang gefiltert
END_VAR
VAR 
	i_Ind: INT;
	f_Summe:REAL;
	timer:ton;
	daten:ARRAY [1..i_Datensaetze] OF REAL;
	Timestruct_to_Time:Timestruct_to_Time;	
	x_Flanke: BOOL;
END_VAR
VAR CONSTANT
	i_Datensaetze:INT:=48;
END_VAR

//Für Aussentemperatur Initialisierung muss x_start gedrückt werden
	 IF x_start  THEN
//Grösse des Array für den Mittelwert bestimmen
		 FOR i_Ind:= 1 TO I_DATENSAETZE DO
			 daten[i_Ind]:= f_AT;
		 END_FOR
	 END_IF
		x_start:=FALSE;
//Timestruct to Time
	timestruct_to_time(t_Ein:=t_time);
//Timer läuft immer
	Timer(IN := NOT Timer.Q, PT :=timestruct_to_time.t_Aus );

	IF Timer.Q THEN
    f_Summe := 0;
//die neuen Temperaturwerte werden ins Array geschrieben
    FOR i_Ind := I_DATENSAETZE TO 2 BY -1  DO
        Daten[i_Ind] := Daten[i_Ind - 1];
        f_Summe := f_Summe + Daten[i_Ind];
    END_FOR
//Rechentemperatur berechnen
    Daten[1] := f_AT;
    f_Summe := f_Summe + f_AT;
    f_Aus:=f_summe / I_DATENSAETZE;
	END_IF

END_FUNCTION_BLOCK

// Math/Minimun
(*Gibt den kleinsten der angeschlossenen Werten aus.
*)
FUNCTION_BLOCK Minimun
(*
Versionsverlauf: 
Version		|Autor	|Bemerkung
------------------------------------------------------------------------------------------------------------ 
17.06.00	|Shgb	|erste Freigabe 
17.06.01	|ShgB	|von Integer auf Real geändert	 
17.08.00	|LeaF	|Freigabe

*)
VAR_INPUT
	f_Ein1 :REAL:=0.00001;//Wert 1
	f_Ein2 :REAL:=0.00001;//Wert 2
	f_Ein3 :REAL:=0.00001;//Wert 3
	f_Ein4 :REAL:=0.00001;//Wert 4
	f_Ein5 :REAL:=0.00001;//Wert 5
	f_Ein6 :REAL:=0.00001;//Wert 6
	f_Ein7 :REAL:=0.00001;//Wert 7
	f_Ein8 :REAL:=0.00001;//Wert 8
END_VAR
VAR_OUTPUT
	f_Aus:REAL;//Kleinste Wert
END_VAR
VAR
	i_Arraypos:INT;
	af_Array: ARRAY [1..8] OF REAL;
END_VAR

// Werte in Array platzieren
	af_Array[1]:=f_Ein1;
	af_Array[2]:=f_Ein2;
	af_Array[3]:=f_Ein3;
	af_Array[4]:=f_Ein4;
	af_Array[5]:=f_Ein5;
	af_Array[6]:=f_Ein6;
	af_Array[7]:=f_Ein7;
	af_Array[8]:=f_Ein8;
		
//Zahlen die grösser als 0 sind
	f_Aus := af_Array[1];	
	
//Auswertung der kleinsten Zahl
	FOR i_Arraypos:=2 TO 8 DO
		IF af_Array[i_Arraypos] <= f_Aus AND af_Array[i_Arraypos] <> 0.00001 THEN
			f_Aus := af_Array[i_Arraypos];
		END_IF
	END_FOR

END_FUNCTION_BLOCK

// Math/Range
(*Wertet aus ob sich der Eingang im angegebenen Bereich befindet. Wert in Grenzen => Ausgang False Wert ausserhalb => Ausgang True
*)
FUNCTION_BLOCK Range
(*
Versionsverlauf: 
Version		|Autor	|Bemerkung
------------------------------------------------------------------------------------------------------------ 
17.06.00	|Shgb	|erste Freigabe  
17.08.00	|LeaF	|Freigabe

*)
VAR_INPUT
	f_Ein:REAL;//Eingang
	f_Min:REAL;//Eingangsbereich Minimum
	f_Max:REAL;//Eingangsbereich Maximum
END_VAR
VAR_OUTPUT
	x_Aus:BOOL;//Ausgang
END_VAR
VAR
END_VAR

x_Aus:= not (f_Ein<=f_Max and f_Ein>=f_Min);

END_FUNCTION_BLOCK

// Math/Timestruct_Kleiner_Gleich_Timestruct
(*Vergleicht zweit Timestructvariablen. Wenn die erste kleiner oder gleich ist wird der Ausgang TRUE andernfalls bleit der Ausgang FALSE
*)
FUNCTION_BLOCK Timestruct_Kleiner_Gleich_Timestruct
(*
Versionsverlauf: 
Version		|Autor	|Bemerkung
------------------------------------------------------------------------------------------------------------ 
17.08.00	|ShgB	|erste Freigabe 

*)
VAR_INPUT
	t_Ein1:TIMESTRUCT;//Referenztimestruct
	t_Ein2:Timestruct;//Vergleichstimestruct
END_VAR
VAR_OUTPUT
	x_Aus:BOOL;//True wenn Vergleichtimestruct kleiner Referenztimestruct ist
END_VAR
VAR
END_VAR

x_Aus:=FALSE;
IF t_Ein1.wDay < t_Ein2.wDay THEN
	x_Aus:=TRUE;
ELSIF t_Ein1.wDay = t_Ein2.wDay THEN
	IF t_Ein1.wHour < t_Ein2.wHour THEN
		x_Aus:=TRUE;
	ELSIF t_Ein1.wHour = t_Ein2.wHour THEN
		IF t_Ein1.wMinute < t_Ein2.wMinute THEN
			x_Aus:=TRUE;
		ELSIF t_Ein1.wMinute = t_Ein2.wMinute THEN
			IF t_Ein1.wSecond < t_Ein2.wSecond THEN
				x_Aus:=TRUE;
			ELSIF t_Ein1.wSecond = t_Ein2.wSecond THEN
				IF t_Ein1.wMilliseconds <= t_Ein2.wMilliseconds THEN
					x_Aus:=TRUE;
				END_IF
			END_IF
		END_IF
	END_IF
END_IF

END_FUNCTION_BLOCK

// Memory/Logger
(*Loggt die angegebenen Datenpunkte im entsprechenden Takt und speichert diese für den angegebenen Zeitraum ab.
*)
FUNCTION_BLOCK Logger
(*
Versionsverlauf: 
Version		|Autor	|Bemerkung
------------------------------------------------------------------------------------------------------------ 
17.07.00	|Shgb	|erste Freigabe  
17.08.00	|LeaF	|Freigabe

*)
VAR_INPUT PERSISTENT
	s_Dir:STRING(255):='C:\TwinCAT\Logger';//Dateipfad für Logdateien
	s_Filename:STRING(255):='Log';//Name der Datei. Wird mit JJJJ_MM_DD ergänzt
	t_Takt:Timestruct := (wSecond := 5);//Takt der Aufzeichnung
	i_Speicherdauer:INT:=14;//Anzahl Tage die gespeichert werden
END_VAR
VAR_INPUT
	x_Ein:BOOL;//Öffent eine Datei und Loggt die Datenpunkte
	x_Record:BOOL;//Datenpunkte werden unabhängig des Taktes geloggts_Titel1:STRING(255);//Titel 1-32 des Datenpunktes
	s_Titel1:STRING(255);//Datenpunkttitel für Kopfzeile
	f_Data1: REAL;//Datenpunkt 1-32
	i_Dezimalstelle1:INT;//Anzahl Dezimalstellen 1-32
	s_Titel2:STRING(255);
	f_Data2: REAL;
	i_Dezimalstelle2:INT;
	s_Titel3:STRING(255);
	f_Data3: REAL;
	i_Dezimalstelle3:INT;
	s_Titel4:STRING(255);
	f_Data4: REAL;
	i_Dezimalstelle4:INT;
	s_Titel5:STRING(255);
	f_Data5: REAL;
	i_Dezimalstelle5:INT;
	s_Titel6:STRING(255);
	f_Data6: REAL;
	i_Dezimalstelle6:INT;
	s_Titel7:STRING(255);
	f_Data7: REAL;
	i_Dezimalstelle7:INT;
	s_Titel8:STRING(255);
	f_Data8: REAL;
	i_Dezimalstelle8:INT;
	s_Titel9:STRING(255);
	f_Data9: REAL;
	i_Dezimalstelle9:INT;
	s_Titel10:STRING(255);
	f_Data10: REAL;
	i_Dezimalstelle10:INT;
	s_Titel11:STRING(255);
	f_Data11: REAL;
	i_Dezimalstelle11:INT;
	s_Titel12:STRING(255);
	f_Data12: REAL;
	i_Dezimalstelle12:INT;
	s_Titel13:STRING(255);
	f_Data13: REAL;
	i_Dezimalstelle13:INT;
	s_Titel14:STRING(255);
	f_Data14: REAL;
	i_Dezimalstelle14:INT;
	s_Titel15:STRING(255);
	f_Data15: REAL;
	i_Dezimalstelle15:INT;
	s_Titel16:STRING(255);
	f_Data16: REAL;
	i_Dezimalstelle16:INT;
	s_Titel17:STRING(255);
	f_Data17: REAL;
	i_Dezimalstelle17:INT;
	s_Titel18:STRING(255);
	f_Data18: REAL;
	i_Dezimalstelle18:INT;
	s_Titel19:STRING(255);
	f_Data19: REAL;
	i_Dezimalstelle19:INT;
	s_Titel20:STRING(255);
	f_Data20: REAL;
	i_Dezimalstelle20:INT;
	s_Titel21:STRING(255);
	f_Data21: REAL;
	i_Dezimalstelle21:INT;
	s_Titel22:STRING(255);
	f_Data22: REAL;
	i_Dezimalstelle22:INT;
	s_Titel23:STRING(255);
	f_Data23: REAL;
	i_Dezimalstelle23:INT;
	s_Titel24:STRING(255);
	f_Data24: REAL;
	i_Dezimalstelle24:INT;
	s_Titel25:STRING(255);
	f_Data25: REAL;
	i_Dezimalstelle25:INT;
	s_Titel26:STRING(255);
	f_Data26: REAL;
	i_Dezimalstelle26:INT;
	s_Titel27:STRING(255);
	f_Data27: REAL;
	i_Dezimalstelle27:INT;
	s_Titel28:STRING(255);
	f_Data28: REAL;
	i_Dezimalstelle28:INT;
	s_Titel29:STRING(255);
	f_Data29: REAL;
	i_Dezimalstelle29:INT;
	s_Titel30:STRING(255);
	f_Data30: REAL;
	i_Dezimalstelle30:INT;
	s_Titel31:STRING(255);
	f_Data31: REAL;
	i_Dezimalstelle31:INT;
	s_Titel32:STRING(255);
	f_Data32: REAL;
	i_Dezimalstelle32:INT;
END_VAR
VAR_OUTPUT
	x_FileOpen:BOOL;//Datei geöffnet
	x_AL_Open:BOOL;//Fehler beim Öffnen der Datei
	x_AL_Write:BOOL;//Fehler beim schreiben der Datenpunkte
	x_AL_Close:BOOL;//Fehler beim Schliessen der Datei
	x_AL_Delete:BOOL;//Fehler beim Löschen der Datei (Datei nicht existent)
END_VAR
VAR
	as_Array:ARRAY[0..33] OF STRING;
	af_Array:ARRAY [1..32] OF REAL;
	ai_Array:ARRAY [1..32] OF INT;
	i_Schrittkette:INT;
	i_Arraypos:INT;
	s_File:STRING;
	s_DelFile:STRING;
	s_temp: STRING;
	s_Data:STRING;
	s_DT: STRING(255);
	f_temp: REAL;
	i_Dezimalzeichen: INT;
	i_LastFile:UINT;
	Timer: TON;
	t_Speicherdauer: TIMESTRUCT;
	Timestruct_to_Time:Timestruct_to_Time;
	FB_CreateDir:FB_CreateDir;
	FB_FileOpen: FB_FileOpen;
	FB_FilePuts: FB_FilePuts;
	FB_FileClose: FB_FileClose;
	FB_FileDelete: FB_FileDelete;
END_VAR
VAR CONSTANT
	I_INIT: INT := 0;
	I_CREATE_DIR: INT := 1;
	I_WAIT_DIR: INT := 2;
	I_FILE_OPEN: INT := 3;
	I_WAIT_OPEN: INT := 4;
	I_FILE_Header: INT := 5;
	I_WAIT_Header: INT := 6;
	I_FILE_WRITE: INT := 7;
	I_END_WRITE: INT := 8;
	I_WAIT_WRITE: INT := 9;
	I_FILE_CLOSE: INT := 10;
	I_WAIT_CLOSE: INT := 11;
END_VAR

//Datenerfassung
	as_Array[0]:='Datum;Zeit;';
	as_Array[1]:=concat(s_Titel1,';');
	as_Array[2]:=concat(s_Titel2,';');
	as_Array[3]:=concat(s_Titel3,';');
	as_Array[4]:=concat(s_Titel4,';');
	as_Array[5]:=concat(s_Titel5,';');
	as_Array[6]:=concat(s_Titel6,';');
	as_Array[7]:=concat(s_Titel7,';');
	as_Array[8]:=concat(s_Titel8,';');
	as_Array[9]:=concat(s_Titel9,';');
	as_Array[10]:=concat(s_Titel10,';');
	as_Array[11]:=concat(s_Titel11,';');
	as_Array[12]:=concat(s_Titel12,';');
	as_Array[13]:=concat(s_Titel13,';');
	as_Array[14]:=concat(s_Titel14,';');
	as_Array[15]:=concat(s_Titel15,';');
	as_Array[16]:=concat(s_Titel16,';');
	as_Array[17]:=concat(s_Titel17,';');
	as_Array[18]:=concat(s_Titel18,';');
	as_Array[19]:=concat(s_Titel19,';');
	as_Array[20]:=concat(s_Titel20,';');
	as_Array[21]:=concat(s_Titel21,';');
	as_Array[22]:=concat(s_Titel22,';');
	as_Array[23]:=concat(s_Titel23,';');
	as_Array[24]:=concat(s_Titel24,';');
	as_Array[25]:=concat(s_Titel25,';');
	as_Array[26]:=concat(s_Titel26,';');
	as_Array[27]:=concat(s_Titel27,';');
	as_Array[28]:=concat(s_Titel28,';');
	as_Array[29]:=concat(s_Titel29,';');
	as_Array[30]:=concat(s_Titel30,';');
	as_Array[31]:=concat(s_Titel31,';');
	as_Array[32]:=concat(s_Titel32,';');
	as_Array[33]:='$N';
	
	af_Array[1]:=f_Data1;
	af_Array[2]:=f_Data2;
	af_Array[3]:=f_Data3;
	af_Array[4]:=f_Data4;
	af_Array[5]:=f_Data5;
	af_Array[6]:=f_Data6;
	af_Array[7]:=f_Data7;
	af_Array[8]:=f_Data8;
	af_Array[9]:=f_Data9;
	af_Array[10]:=f_Data10;
	af_Array[11]:=f_Data11;
	af_Array[12]:=f_Data12;
	af_Array[13]:=f_Data13;
	af_Array[14]:=f_Data14;
	af_Array[15]:=f_Data15;
	af_Array[16]:=f_Data16;
	af_Array[17]:=f_Data17;
	af_Array[18]:=f_Data18;
	af_Array[19]:=f_Data19;
	af_Array[20]:=f_Data20;
	af_Array[21]:=f_Data21;
	af_Array[22]:=f_Data22;
	af_Array[23]:=f_Data23;
	af_Array[24]:=f_Data24;
	af_Array[25]:=f_Data25;
	af_Array[26]:=f_Data26;
	af_Array[27]:=f_Data27;
	af_Array[28]:=f_Data28;
	af_Array[29]:=f_Data29;
	af_Array[30]:=f_Data30;
	af_Array[31]:=f_Data31;
	af_Array[32]:=f_Data32;
	
	ai_Array[1]:=i_Dezimalstelle1;
	ai_Array[2]:=i_Dezimalstelle2;
	ai_Array[3]:=i_Dezimalstelle3;
	ai_Array[4]:=i_Dezimalstelle4;
	ai_Array[5]:=i_Dezimalstelle5;
	ai_Array[6]:=i_Dezimalstelle6;
	ai_Array[7]:=i_Dezimalstelle7;
	ai_Array[8]:=i_Dezimalstelle8;
	ai_Array[9]:=i_Dezimalstelle9;
	ai_Array[10]:=i_Dezimalstelle10;
	ai_Array[11]:=i_Dezimalstelle11;
	ai_Array[12]:=i_Dezimalstelle12;
	ai_Array[13]:=i_Dezimalstelle13;
	ai_Array[14]:=i_Dezimalstelle14;
	ai_Array[15]:=i_Dezimalstelle15;
	ai_Array[16]:=i_Dezimalstelle16;
	ai_Array[17]:=i_Dezimalstelle17;
	ai_Array[18]:=i_Dezimalstelle18;
	ai_Array[19]:=i_Dezimalstelle19;
	ai_Array[20]:=i_Dezimalstelle20;
	ai_Array[21]:=i_Dezimalstelle21;
	ai_Array[22]:=i_Dezimalstelle22;
	ai_Array[23]:=i_Dezimalstelle23;
	ai_Array[24]:=i_Dezimalstelle24;
	ai_Array[25]:=i_Dezimalstelle25;
	ai_Array[26]:=i_Dezimalstelle26;
	ai_Array[27]:=i_Dezimalstelle27;
	ai_Array[28]:=i_Dezimalstelle28;
	ai_Array[29]:=i_Dezimalstelle29;
	ai_Array[30]:=i_Dezimalstelle30;
	ai_Array[31]:=i_Dezimalstelle31;
	ai_Array[32]:=i_Dezimalstelle32;
	

//Dateiname erstellen
	s_File:=CONCAT(STR1:=s_Dir, STR2:='\');
	s_File:=CONCAT(STR1:=s_File, STR2:=s_Filename);
	s_File:=CONCAT(STR1:=s_File, STR2:='_');
	s_File:=CONCAT(STR1:=s_File, STR2:=DWORD_TO_STRING(Globale_Uhr.systemtimestruct.wYear));
	s_File:=CONCAT(STR1:=s_File, STR2:='_');
	s_File:=CONCAT(STR1:=s_File, STR2:=DWORD_TO_STRING(Globale_Uhr.systemtimestruct.wMonth));
	s_File:=CONCAT(STR1:=s_File, STR2:='_');
	s_File:=CONCAT(STR1:=s_File, STR2:=DWORD_TO_STRING(Globale_Uhr.systemtimestruct.wDay));
	s_File:=CONCAT(STR1:=s_File, STR2:='.csv');

//Pfad für zu löschende Datei
	t_Speicherdauer:=DT_TO_SYSTEMTIME( Globale_Uhr.systemDateAndTime-i_Speicherdauer*T#1D-T#1D);
				
	s_DelFile:=CONCAT(STR1:=s_Dir, STR2:='\');
	s_DelFile:=CONCAT(STR1:=s_DelFile, STR2:=s_Filename);
	s_DelFile:=CONCAT(STR1:=s_DelFile, STR2:='_');
	s_DelFile:=CONCAT(STR1:=s_DelFile, STR2:=DWORD_TO_STRING(t_Speicherdauer.wYear));
	s_DelFile:=CONCAT(STR1:=s_DelFile, STR2:='_');
	s_DelFile:=CONCAT(STR1:=s_DelFile, STR2:=DWORD_TO_STRING(t_Speicherdauer.wMonth));
	s_DelFile:=CONCAT(STR1:=s_DelFile, STR2:='_');
	s_DelFile:=CONCAT(STR1:=s_DelFile, STR2:=DWORD_TO_STRING(t_Speicherdauer.wDay));
	s_DelFile:=CONCAT(STR1:=s_DelFile, STR2:='.csv');

//Datum und Uhrzeit erstellen
	s_DT:='';
	s_DT:=CONCAT(STR1:=s_DT, STR2:=DWORD_TO_STRING(Globale_Uhr.systemtimestruct.wDay));
	s_DT:=CONCAT(STR1:=s_DT, STR2:='.');
	s_DT:=CONCAT(STR1:=s_DT, STR2:=DWORD_TO_STRING(Globale_Uhr.systemtimestruct.wMonth));
	s_DT:=CONCAT(STR1:=s_DT, STR2:='.');
	s_DT:=CONCAT(STR1:=s_DT, STR2:=DWORD_TO_STRING(Globale_Uhr.systemtimestruct.wYear));
	s_DT:=CONCAT(STR1:=s_DT, STR2:=';');
	s_DT:=CONCAT(STR1:=s_DT, STR2:=DWORD_TO_STRING(Globale_Uhr.systemtimestruct.wHour));
	s_DT:=CONCAT(STR1:=s_DT, STR2:=':');
	s_DT:=CONCAT(STR1:=s_DT, STR2:=DWORD_TO_STRING(Globale_Uhr.systemtimestruct.wMinute));
	s_DT:=CONCAT(STR1:=s_DT, STR2:=':');
	s_DT:=CONCAT(STR1:=s_DT, STR2:=DWORD_TO_STRING(Globale_Uhr.systemtimestruct.wSecond));			

//Timestruct to Time
	Timestruct_to_Time(t_Ein:=t_Takt);
	
//Takt
	Timer(IN:= x_Ein AND NOT Timer.Q, PT:= Timestruct_to_Time.t_Aus);
	
//Case
	CASE i_Schrittkette OF
		I_INIT:
			IF x_Ein THEN
				i_Schrittkette:=I_CREATE_DIR;
			END_IF
		
		I_CREATE_DIR:
			FB_CreateDir.bExecute:=TRUE;
			i_Schrittkette:=I_WAIT_DIR;
	
		I_WAIT_DIR:
			IF NOT FB_CreateDir.bBusy THEN
				i_Schrittkette:=I_FILE_OPEN;
				FB_CreateDir.bExecute:=FALSE;
			END_IF
		
		I_FILE_OPEN:
			FB_FileOpen.sPathName:=s_File;
			FB_FileOpen.bExecute:=TRUE;
			i_Schrittkette:= I_WAIT_OPEN;
			
		I_WAIT_OPEN:
			IF NOT FB_FileOpen.bBusy AND FB_FileOpen.hFile <> 0 AND FB_FileOpen.hFile <> i_LastFile THEN
				IF s_File <> s_temp THEN
					i_Schrittkette:=I_FILE_Header;
					FB_FileDelete.bExecute:=TRUE;
					s_temp:=s_File;
				ELSE
					i_Schrittkette:=I_WAIT_WRITE;
					FB_FileDelete.bExecute:=FALSE;	
				END_IF
				i_Arraypos:=0;
				FB_FileOpen.bExecute:=FALSE;
			END_IF
			IF NOT FB_FileOpen.bBusy AND (FB_FileOpen.hFile = 0 OR FB_FileOpen.hFile = i_LastFile)  THEN
				i_Schrittkette:=I_FILE_OPEN;
				FB_FileOpen.bExecute:=FALSE;
			END_IF
			
		I_FILE_Header:
			FB_FilePuts.sLine:=as_Array[i_Arraypos];
			IF LEN(as_Array[i_Arraypos])>0 THEN 
				FB_FilePuts.bExecute:=TRUE;
			END_IF
			i_Schrittkette:= I_WAIT_Header;
			i_Arraypos:=i_Arraypos+1;
		
		I_WAIT_Header:
			IF NOT FB_FilePuts.bBusy AND i_Arraypos <=33 THEN
				i_Schrittkette:=I_FILE_Header;
				FB_FilePuts.bExecute:=FALSE;
			END_IF
			IF NOT FB_FilePuts.bBusy AND i_Arraypos =34 THEN
				i_Schrittkette:=I_WAIT_WRITE;
				i_Arraypos:=0;
				FB_FilePuts.bExecute:=FALSE;
			END_IF
						
		I_WAIT_WRITE:
			IF NOT FB_FilePuts.bBusy AND i_Arraypos<=33 THEN
				i_Schrittkette:=I_FILE_WRITE;
				FB_FilePuts.bExecute:=FALSE;
			END_IF
			IF NOT FB_FilePuts.bBusy AND i_Arraypos>33 THEN
				i_Schrittkette:=I_END_WRITE;
				i_Arraypos:=0;
				FB_FilePuts.bExecute:=FALSE;
			END_IF
		
		I_FILE_WRITE:
			CASE i_Arraypos OF
				0:
					FB_FilePuts.sLine:=concat(STR1:= s_DT,STR2:=';');
				
				1..32:
					s_Data:='';
					s_Data:=CONCAT(STR1:=s_Data,STR2:=DINT_TO_STRING(TRUNC(af_Array[i_Arraypos])));
					IF ai_Array[i_Arraypos] >0 THEN
						s_Data:=CONCAT(STR1:=s_Data, STR2:='.');
						f_temp:=af_Array[i_Arraypos]-TRUNC(af_Array[i_Arraypos]);
						FOR i_Dezimalzeichen:=1 TO ai_Array[i_Arraypos] DO
							f_temp:=f_temp*10;
						END_FOR
					s_Data:=CONCAT(STR1:=s_Data,STR2:=DINT_TO_STRING(TRUNC(f_temp)));
					END_IF
					s_Data:=CONCAT(STR1:=s_Data, STR2:=';');
					FB_FilePuts.sLine:=s_Data;				
				
				33:
					FB_FilePuts.sLine:='$N';
			END_CASE
			IF LEN(as_Array[i_Arraypos])>0 THEN 
				FB_FilePuts.bExecute:=TRUE;
			END_IF
			i_Schrittkette:= I_WAIT_WRITE;
			i_Arraypos:=i_Arraypos+1;	

		I_END_WRITE:
			IF Timer.Q THEN
				i_Schrittkette:=I_FILE_WRITE;
			END_IF
			
			IF NOT x_Ein OR s_File <> s_temp THEN
				i_Schrittkette:=I_FILE_CLOSE;
			END_IF	
			
		I_FILE_CLOSE:
			FB_FileClose.bExecute:=TRUE;
			i_Schrittkette:= I_WAIT_CLOSE;
			
		I_WAIT_CLOSE:
			IF NOT FB_FileClose.bBusy THEN
				FB_FileClose.bExecute:=FALSE;
				i_LastFile:=FB_FileOpen.hFile;
				i_Schrittkette:=I_INIT;
			END_IF
	END_CASE

//FB Create Dir
	FB_CreateDir(
		sPathName:= s_Dir);
				
//FB File Open
	FB_FileOpen( 
		nMode:= FOPEN_MODEAPPEND OR FOPEN_MODEPLUS,
		bError=> x_AL_Open);
		
//FB File Write
	FB_FilePuts( 
				hFile:= FB_FileOpen.hFile,
				bError=> x_AL_Write);
				
//FB File Close
	FB_FileClose(
				hFile:= FB_FileOpen.hFile,
				bError=> x_AL_Close);
				
//File Open
	x_FileOpen:=i_Schrittkette>=I_WAIT_Header;
	
//FB Delete File
	FB_FileDelete( 
		sPathName:= s_DelFile, 
		bError=> x_AL_Delete);

END_FUNCTION_BLOCK

// Regler/EEV
(*Dieser Funktionsbaustein regelt die Verdampfungstemperatur, mittels EEV, um den Überhitzungssollwert tiefer als die Sauggastemperatur.
Formel: Soll Verdampfung = Sauggastemperatur - Überhitzungssollwert
Die Soll Verdampfung wird zudem noch durch den MOP begrenzt. Ist die Überhitzung länger als 2 Minuten unterhalb von 2K so wird ein Alarm ausgelöst.
*)
FUNCTION_BLOCK EEV
(*
Versionsverlauf: 
Version		|Autor	|Bemerkung
------------------------------------------------------------------------------------------------------------ 
17.06.00	|Shgb	|erste Freigabe 
17.06.01	|ShgB	|von Integer auf Real geändert	
17.06.02	|ShgB	|Von Time auf Timestruct geändert
17.08.00	|LeaF	|Freigabe

*)
VAR_INPUT
	x_Enable:BOOL;//Regelung Freigeben
	x_Quittieren:BOOL;//Alarme quittieren
	f_Verdampfunstemperatur:REAL;//Verdampfungstemperatur
	f_Sauggastemperatur:REAL;//Sauggastemperatur
	x_SW_Reset:BOOL;//Setzt die Standardwerte für den Kompressorty zurück
	f_MOP_Einsatzgrenzen: REAL := 0.00001;//Dynamischer MOP von Einsatzgrenzen
	dut_Kompressortyp:SW_Einsatzgrenzen:=SW_ALZ.Bitzer_Scroll_R410a;//Kompressortyp als DUT Angabe Standard Bitzer Scroll 410a
END_VAR
VAR_INPUT PERSISTENT
	f_SollwertUBH:REAL := 6;//Sollwert für die Überhitzung
	f_MOP:REAL;//Maximal Operating Pressure
	f_PFaktor:REAL:=3.0;//P Faktor für Regelung
	f_IFaktor:REAL:=0.05;//I Faktor für Regelung
	f_DFaktor:REAL:=0;//D Faktor für Regelung
	t_Takt:timestruct := (wMilliseconds := 100);//Berechnungstakt des PID Reglers
	f_MinUBH:REAL:=2;//Minimale Überhitzung
	t_AL_EEV:Timestruct := (wMinute := 2);//Zeit bis Alarm ausgelöst wird
END_VAR
VAR_OUTPUT
	f_UBH:REAL;//Berechnete Überhitzung
	f_Regelsignal:REAL;//Regelsignal für das Expansionsventil
	x_Alarm:BOOL;//Überhitzung wurde nicht erreicht/
END_VAR
VAR
	f_SollVerdampfung:REAL;
	PID: PIDRegler;
	UBH_Timer: TON;
	x_TempAlarm: BOOL;
	Timestruct_to_Time: Timestruct_to_Time;
END_VAR

VAR PERSISTENT
	x_Laden: BOOL;//Variable ist beim ersten aufstarten False und lädt somit die eingestellten Daten
END_VAR

//Überhitzung 
	f_UBH:=f_Sauggastemperatur-f_Verdampfunstemperatur;
	
//Soll Verdampfungstemperatur berechnen
	f_SollVerdampfung:=f_Sauggastemperatur-f_SollwertUBH;
	//MOP 
	IF f_SollVerdampfung > f_MOP_Einsatzgrenzen AND f_MOP_Einsatzgrenzen <> 0.00001 THEN
		f_SollVerdampfung:=f_MOP_Einsatzgrenzen;
	END_IF
	
	IF f_SollVerdampfung > f_MOP THEN
		f_SollVerdampfung:=f_MOP;
	END_IF
	
//PID Regelung
	PID(
		x_Enable:= x_Enable and not x_Alarm, 
		x_Invertiert:= FALSE, 
		x_Manuell:= FALSE, 
		f_Sollwert:= f_SollVerdampfung, 
		f_Ist:= f_Verdampfunstemperatur, 
		f_Offset:= 0, 
		f_Min:= 0, 
		f_Max:= 100, 
		f_Manuell:= 0, 
		f_PFaktor:= f_PFaktor, 
		f_IFaktor:= f_IFaktor, 
		f_DFaktor:= f_DFaktor, 
		t_Takt:= t_Takt, 
		f_Regelsignal=> f_Regelsignal);
		
//Überhitzungsschutz < 2K
	IF f_UBH < f_MinUBH THEN
		f_Regelsignal:=f_Regelsignal/2;
	END_IF

//Alarm
	IF x_Quittieren THEN
		x_Alarm:=FALSE;
	END_IF
	
	//Timestruct to Time
	Timestruct_to_Time(t_Ein:= t_AL_EEV);
	
	UBH_Timer(IN:= f_UBH<2.0 AND x_Enable, PT:= Timestruct_to_Time.t_Aus, Q=> x_TempAlarm, ET=> );
	
	IF x_TempAlarm THEN
		x_Alarm:=TRUE;
	END_IF	
	
//Reset Sollwerte
	IF x_SW_Reset OR NOT x_Laden THEN
		f_MOP:=dut_Kompressortyp.f_SW_EG_MaxVerd-2;
		x_Laden:=TRUE;
	END_IF

END_FUNCTION_BLOCK

// Verdichter/Einsatzgrenzen
(*Überwacht die Einsatzgrenzen der Kompressoren und gibt mit einem BOOL an ob diese sich noch in den Einsatzgrenzen befinden. Ein Toleranzband kann zusätzlich mit einer Zeit bestimmt werden.
Verlässt der Kompressor die Einsatzgrenzen ober wird zu lange im Toleranzband betrieben so wird das Ausgangsbool auf FALSE gesetzt. Für weitere Infos siehe Beschrieb im FB.
*)
FUNCTION_BLOCK Einsatzgrenzen
(*
Versionsverlauf: 
Version		|Autor	|Bemerkung
------------------------------------------------------------------------------------------------------------ 
17.06.00	|Shgb	|erste Freigabe 
17.06.01	|ShgB	|von Integer auf Real geändert
17.06.02	|ShgB	|Von Time auf Timestruct geändert
17.07.00	|ShgB	|MOP Berechnung angepasst

		  F	_____________5__________ E
		  /							\ 4
	  6	/							 \ D
	  /								 | 3
  G /								 | C
	|								/  
	|							  /
  7 |							/ 2
	|_________________________/
	A			1			  B
*)
VAR_INPUT 
	f_Verd:REAL;//Aktuelle Verdampfungstemperatur
	f_Kond:REAL;//Aktuelle Kondensationstemperatur
	x_Betriebsmeldung: BOOL;//Sobald die Betriebsmeldung kommt wird die Auswertung um die eingestellte Verzögert aktiv
	x_Quittieren: BOOL;//Alarme quittieren
	x_SW_Reset:BOOL;//Setzt die Standardwerte für den Kompressorty zurück
	dut_Kompressortyp:SW_Einsatzgrenzen:=SW_ALZ.Bitzer_Scroll_R410a;//Kompressortyp als DUT Angabe Standard Bitzer Scroll 410a
END_VAR
VAR_INPUT PERSISTENT
	f_MinVerd:REAL;//Minimale Verdampfungstemperatur Linie 7
	f_MaxVerd:REAL;//Maximale Verdampfungstemperatur Linie 3
	f_MinKond:REAL;//Minimale Kondensationstemperatur Punkt A
	f_MaxKond:REAL;//Maximale Kondensationstemperatur Linie 5
	f_BVerd:REAL;//Verdampfungstemperatur beim Punkt B
	f_BKond:REAL;//Kondensationstemperatur beim Punkt B
	f_CKond:REAL;//Kondensationstemperatur beim Punkt C
	f_DKond:REAL;//Kondensationstemperatur beim Punkt D
	f_EVerd:REAL;//Verdampfungstemperatur beim Punkt E
	f_FVerd:REAL;//Verdampfungstemperatur beim Punkt F
	f_GKond:REAL;//Kondensationstemperatur beim Punkt G
	f_Toleranz:REAL:=1;//Breite des Toleranzbandes in °C
	t_Toleranz:timestruct := (wMinute := 5);//Zeit die der Kompressor im Toleranzband sein darf
	f_GUI_Zoom:REAL;//Zoomfaktor für das Vergrössern der Grafik
	i_GUI_VersatzX:INT;//Versatz der Grafik in X Richtung (Verdampfung)
	i_GUI_VersatzY:INT;//Versatz der Grafik in Y Richtung (Kondensation)
END_VAR
VAR_OUTPUT
	f_ActMinKond:REAL;//Aktuelle mindest Kondensation laut Einsatzgrenzendiagramm
	f_ActMaxKond:REAL;//Aktuelle maximale Kondensation laut Einsatzgrenzendiagramm
	f_ActMinVerd:REAL;//Aktuelle mindest Verdampfung laut Einsatgrenzendiagramm
	f_ActMaxVerd:REAL;//Aktuelle maximale Verdampfung laut Einsatzgrenzendiagramm
	x_Aus:BOOL;//Befindet sich der Kompressor in den Einsatzgrenzen
	x_BM_ND:BOOL;//Kompressor befindet sich im Toleranzband auf der Niederdruckseite
	x_AL_ND:BOOL;//Kompressor ist ausserhalb der Einsatzgrenzen auf der Niederdruckseite
	x_BM_HD:BOOL;//Kompressor befindet sich im Toleranzband auf der Hochdruckseite
	x_AL_HD:BOOL;//Kompressor ist ausserhalb der Einsatzgrenzen auf der Hochdruckseite
	x_BM_MOP: BOOL;//Kompressor befindet sich im Toleranzband vor dem MOP Alarm
	x_AL_MOP: BOOL;//MOP wurde überschritten
END_VAR
VAR
	Timer: TON;
	x_Timer:BOOL;
	Maximum: Maximum;
	Linie1_Verd: Converter2Punkt;
	Linie1_Kond: Converter2Punkt;
	Linie2_Verd: Converter2Punkt;
	Linie2_Kond: Converter2Punkt;
	Linie4_Kond: Converter2Punkt;
	Linie4_Verd: Converter2Punkt;
	Linie6_Verd: Converter2Punkt;
	Linie6_Kond: Converter2Punkt;
	Minimum: Minimun;
	t_Temp: TIME;
	Timestruct_to_Time:Timestruct_to_Time;
	FB_MIN_KD: maximum;
	FB_MIN_VD: maximum;
	FB_MAX_KD: Minimun;
	FB_MAX_VD: Minimun;
	Betriebsmeldung:Ton;
END_VAR
VAR PERSISTENT
	x_Laden:BOOL;//Variable ist beim ersten aufstarten False und lädt somit die eingestellten Daten
END_VAR
VAR//Variablen für Grafik
	f_GUI_Verd:REAL;//Aktuelle Verdampfungstemperatur
	f_GUI_Kond:REAL;//Aktuelle Kondensationstemperatur
	f_GUI_MinVerd:REAL;//Minimale Verdampfungstemperatur Linie 7
	f_GUI_MaxVerd:REAL;//Maximale Verdampfungstemperatur Linie 3
	f_GUI_MinKond:REAL;//Minimale Kondensationstemperatur Punkt A
	f_GUI_MaxKond:REAL;//Maximale Kondensationstemperatur Linie 5
	f_GUI_BVerd:REAL;//Verdampfungstemperatur beim Punkt B
	f_GUI_BKond:REAL;//Kondensationstemperatur beim Punkt B
	f_GUI_CKond:REAL;//Kondensationstemperatur beim Punkt C
	f_GUI_DKond:REAL;//Kondensationstemperatur beim Punkt D
	f_GUI_EVerd:REAL;//Verdampfungstemperatur beim Punkt E
	f_GUI_FVerd:REAL;//Verdampfungstemperatur beim Punkt F
	f_GUI_GKond:REAL;//Kondensationstemperatur beim Punkt G
END_VAR

//Linienberechnungen
	//Linie 1
		Linie1_Verd(
			f_Ein:= f_Verd, 
			f_Ein_Min:= f_MinVerd, 
			f_Ein_Max:= f_BVerd, 
			f_Aus_Min:= f_MinKond, 
			f_Aus_Max:= f_BKond);
			
		Linie1_Kond(
			f_Ein:= f_Kond, 
			f_Ein_Min:= f_MinKond, 
			f_Ein_Max:= f_BKond, 
			f_Aus_Min:= f_MinVerd, 
			f_Aus_Max:= f_BVerd);
			
	//Linie 2
		Linie2_Verd(
			f_Ein:= f_Verd, 
			f_Ein_Min:= f_BVerd, 
			f_Ein_Max:= f_MaxVerd, 
			f_Aus_Min:= f_BKond, 
			f_Aus_Max:= f_CKond);
			
		Linie2_Kond(
			f_Ein:= f_Kond, 
			f_Ein_Min:= f_BVerd, 
			f_Ein_Max:= f_MaxVerd, 
			f_Aus_Min:= f_BKond, 
			f_Aus_Max:= f_CKond);
			
	//Linie 4
		Linie4_Kond(
			f_Ein:= f_Kond, 
			f_Ein_Min:= f_MaxKond, 
			f_Ein_Max:= f_DKond, 
			f_Aus_Min:= f_EVerd, 
			f_Aus_Max:= f_MaxVerd);
			
		Linie4_Verd(
			f_Ein:= f_Verd, 
			f_Ein_Min:= f_EVerd, 
			f_Ein_Max:= f_MaxVerd, 
			f_Aus_Min:= f_MaxKond, 
			f_Aus_Max:= f_DKond);
			
	//Linie 6
		Linie6_Verd(
			f_Ein:= f_Verd, 
			f_Ein_Min:= f_MinVerd, 
			f_Ein_Max:= f_FVerd, 
			f_Aus_Min:= f_GKond, 
			f_Aus_Max:= f_MaxKond);
				
		Linie6_Kond(
			f_Ein:= f_Kond, 
			f_Ein_Min:= f_GKond, 
			f_Ein_Max:= f_MaxKond, 
			f_Aus_Min:= f_MinVerd, 
			f_Aus_Max:= f_FVerd);
			
//Minimale Kondensationstemperatur wird durch die Linien 1,  2 und f_MinKond vom Einsatzgrenzendiagramm gegeben. Die höhere von beiden wird genommen.
	FB_MIN_KD(
		f_Ein1:= Linie1_Verd.f_Aus, 
		f_Ein2:= Linie2_Verd.f_Aus, 
		f_Ein3:= f_MinKond, 
		f_Aus=> f_ActMinKond);
			
//Maximale Kondensationstemperaturwird durch Linie 4, 6 und f_MaxKond vom Einsatzgrenzendiagramm gegeben. Die kleinere von den dreien wird genommen. Linie 5 ist f_MaxKond
	FB_MAX_KD(
		f_Ein1:=Linie4_Verd.f_Aus,
		f_Ein2:=Linie6_Verd.f_Aus,
		f_Ein3:=f_MaxKond,
		f_Aus=>f_ActMaxKond);
			
//Minimale Verdampfungstemperatur durch Linie 6 und f_MinVerd gegeben
	FB_MIN_VD(
		f_Ein1:=Linie6_Kond.f_Aus,
		f_Ein2:= f_MinVerd,
		f_Aus=>f_ActMinVerd);
				
//Maximale Verdampfungstemperatur 
	IF f_Kond <= f_BKond AND f_Kond>= f_MinKond THEN
		f_ActMaxVerd:=Linie1_Kond.f_Aus;
	ELSE
		FB_MAX_VD(
			f_Ein1:=Linie2_Kond.f_Aus,
			f_Ein2:=Linie4_Kond.f_Aus,
			f_Ein3:=f_MaxVerd,
			f_Aus=>f_ActMaxVerd);
	END_IF

//TImestruct to Time
	Timestruct_to_Time(t_Ein:=t_Toleranz);
	
//Auswertung ob in den Einsatzgrenzen mit Timer
	Betriebsmeldung(IN:=x_Betriebsmeldung,PT:=Timestruct_to_Time.t_Aus);

	Timer(IN:= f_Verd < f_ActMinVerd+f_Toleranz OR
		f_Verd > f_ActMaxVerd-f_Toleranz OR
		f_Kond < f_ActMinKond+f_Toleranz OR
		f_Kond > f_ActMaxKond-f_Toleranz, PT:= Timestruct_to_Time.t_Aus, Q=> x_Timer, ET=> );
			
	x_Aus :=NOT Betriebsmeldung.Q OR(f_Verd > f_ActMinVerd AND
		f_Verd < f_ActMaxVerd AND
		f_Kond > f_ActMinKond AND
		f_Kond < f_ActMaxKond AND
		NOT x_Timer);

//Alarme
	IF x_Quittieren THEN
		x_AL_HD := FALSE;
		x_AL_ND := FALSE;
		x_AL_MOP:= FALSE;
	END_IF

	x_BM_ND:=f_Verd<f_ActMinVerd+f_Toleranz;
		
	IF f_Verd<f_ActMinVerd THEN
		x_AL_ND:=TRUE;
	END_IF
		
	x_BM_HD:=f_Kond>f_ActMaxKond-f_Toleranz;
		
	IF f_Kond>f_ActMaxKond THEN
		x_AL_HD:=TRUE;
	END_IF
	
	x_BM_MOP:=f_Verd>f_ActMaxVerd-f_Toleranz;
	
	IF f_Verd>f_ActMaxVerd THEN
		x_AL_MOP:=TRUE;
	END_IF
	
//Reset Sollwerte
	IF x_SW_Reset OR not x_Laden THEN
		f_MinVerd:=dut_Kompressortyp.f_SW_EG_MinVerd;
		f_MaxVerd:=dut_Kompressortyp.f_SW_EG_MaxVerd;
		f_MinKond:=dut_Kompressortyp.f_SW_EG_MinKond;
		f_MaxKond:=dut_Kompressortyp.f_SW_EG_MaxKond;
		f_BVerd:=dut_Kompressortyp.f_SW_EG_BVerd;
		f_BKond:=dut_Kompressortyp.f_SW_EG_BKond;
		f_CKond:=dut_Kompressortyp.f_SW_EG_CKond;
		f_DKond:=dut_Kompressortyp.f_SW_EG_DKond;
		f_EVerd:=dut_Kompressortyp.f_SW_EG_EVerd;
		f_FVerd:=dut_Kompressortyp.f_SW_EG_FVerd;
		f_GKond:=dut_Kompressortyp.f_SW_EG_GKond;
		x_Laden:=TRUE;
	END_IF
	
//GUI Anpassungen
	f_GUI_Verd:=f_Verd*f_GUI_Zoom+i_GUI_VersatzX;
	f_GUI_Kond:=f_Kond*f_GUI_Zoom+i_GUI_VersatzY*-1;
	f_GUI_MinVerd:=f_MinVerd*f_GUI_Zoom+i_GUI_VersatzX;
	f_GUI_MaxVerd:=f_MaxVerd*f_GUI_Zoom+i_GUI_VersatzX;
	f_GUI_MinKond:=f_MinKond*f_GUI_Zoom+i_GUI_VersatzY*-1;
	f_GUI_MaxKond:=f_MaxKond*f_GUI_Zoom+i_GUI_VersatzY*-1;
	f_GUI_BVerd:=f_BVerd*f_GUI_Zoom+i_GUI_VersatzX;
	f_GUI_BKond:=f_BKond*f_GUI_Zoom+i_GUI_VersatzY*-1;
	f_GUI_CKond:=f_CKond*f_GUI_Zoom+i_GUI_VersatzY*-1;
	f_GUI_DKond:=f_DKond*f_GUI_Zoom+i_GUI_VersatzY*-1;
	f_GUI_EVerd:=f_EVerd*f_GUI_Zoom+i_GUI_VersatzX;
	f_GUI_FVerd:=f_FVerd*f_GUI_Zoom+i_GUI_VersatzX;
	f_GUI_GKond:=f_GKond*f_GUI_Zoom+i_GUI_VersatzY*-1;

END_FUNCTION_BLOCK

// Regler/PIDRegler
(*Der PID Regler rechnet die Differenz zwischen dem Sollwert und dem Istwert aus und multipliziert diese mit dem P Faktor. 
Die I und D Anteile werden bei jedem Takt neu berechnet und auf den P Anteil dazu addiert. 
Je grösser die Faktoren sind, desto schneller und instabiler wirde der Regler.
P Anteil: 
Formel Normal: (Sollwert + Ossfet - Istwert) x P Faktor 
Formel Invertiert: (Istwert - Sollwert - Offset) x P Faktor 
I Anteil: 
Formel: I Anteil + I Faktor x P Anteil 
D Anteil: 
Formel: (P Anteil - P Anteil (vom letzten Takt)) x D Faktor
Regelsignal: P + I + D Anteil
*)
FUNCTION_BLOCK PIDRegler
(*
Versionsverlauf: 
Version		|Autor	|Bemerkung
------------------------------------------------------------------------------------------------------------ 
17.06.00	|Shgb	|erste Freigabe 
17.06.01	|ShgB	|von Integer auf Real geändert	
17.06.02	|ShgB	|Von Time auf Timestruct geändert
17.07.00	|ShgB	|Offset und Invertierung geändert.
17.08.00	|LeaF	|Freigabe	

*)
VAR_INPUT
	x_Enable:BOOL;//Freigabe des Reglers
	f_Ist:REAL;//Istwert
END_VAR
VAR_INPUT PERSISTENT
	x_Invertiert:BOOL;//Bei Kühlfunktionen aktiv
	x_Manuell:BOOL;//Manuelles Regelsignal aktivieren
	f_Sollwert:REAL;//Sollwertvorgabe
	f_Offset:REAL;//Offset
	f_Min:REAL;//Minimales Regelsignal
	f_Max:REAL;//Maximales Regelsignal
	f_Manuell:REAL;//Manuelles Regelsignal
	f_PFaktor:REAL;//Proportionalfaktor
	f_IFaktor:REAL;//Integralfaktor
	f_DFaktor:REAL;//Differenzialfaktor
	t_Takt:timestruct;//Regelungstakt
END_VAR
VAR_OUTPUT
	f_Regelsignal:REAL;//Regelsignal
END_VAR
VAR
	f_IAnteil,f_ISpeicher,f_DAnteil:REAL;
	f_PAnteil,f_DSpeicher:REAL;
	P_Anteil: PRegler;
	Timer: TON;
	x_Takt:BOOL;
	Timestruct_to_Time: Timestruct_to_Time;
END_VAR

//P Anteil	
	P_Anteil(
		x_Enable:= x_Enable, 
		x_Invertiert:= x_Invertiert, 
		x_Manuell:= FALSE, 
		f_Sollwert:= f_Sollwert, 
		f_Ist:= f_Ist, 
		f_Offset:= f_Offset, 
		f_Min:= -f_Max, 
		f_Max:= f_Max, 
		f_Manuell:= 0, 
		f_PFaktor:= f_PFaktor, 
		f_Regelsignal=> f_PAnteil);
		
//TImestruct to Time
	Timestruct_to_Time(t_Ein:=t_Takt);	

//Takt
	Timer(IN:= x_Enable AND NOT x_Takt, PT:= Timestruct_to_Time.t_Aus, Q=> x_Takt, ET=> );
	
//I Anteil
	IF x_Takt AND f_Regelsignal<f_Max AND f_Regelsignal>f_Min THEN
		f_ISpeicher:=f_ISpeicher+f_IFaktor*f_PAnteil;
	END_IF

//D Anteil
	IF x_Takt THEN
		f_DAnteil:=(f_PAnteil-f_DSpeicher)*f_DFaktor;
		f_DSpeicher:=f_PAnteil;
	END_IF

//Reset Speicher
	IF NOT x_Enable THEN
		f_ISpeicher:=0.0;
		f_DSpeicher:=0.0;
	END_IF

//Grenzen einhalten	
	f_Regelsignal := LIMIT(f_Min,f_ISpeicher+f_DAnteil+f_PAnteil, f_Max);

//Manuell	
	IF x_Manuell THEN
		f_Regelsignal:=f_Manuell;
	END_IF

END_FUNCTION_BLOCK

// Regler/PRegler
(*Der P Regler rechnet die Differenz zwischen dem Sollwert und dem Istwert aus und multipliziert diese mit dem P Faktor. Je grösser der Faktor ist, desto schneller und instabiler wirde der Regler.
Formel Normal: (Sollwert + Ossfet - Istwert) x P Faktor 
Formel Invertiert: (Istwert - Sollwert - Offset) x P Faktor 
*)
FUNCTION_BLOCK PRegler
(*
Versionsverlauf: 
Version		|Autor	|Bemerkung
------------------------------------------------------------------------------------------------------------ 
17.06.00	|Shgb	|erste Freigabe 
17.06.01	|ShgB	|von Integer auf Real geändert	
17.07.00	|ShgB	|Offset und Invertierung geändert.	
17.08.00	|LeaF	|Freigabe

*)
VAR_INPUT
	x_Enable:BOOL;//Freigabe des Reglers
	f_Ist:REAL;//Istwert
END_VAR
VAR_INPUT PERSISTENT
	x_Invertiert:BOOL;//Bei Kühlfunktionen aktiv
	x_Manuell:BOOL;//Manuelles Regelsignal aktivieren
	f_Sollwert:REAL;//Sollwertvorgabe
	f_Offset:REAL;//Offset
	f_Min:REAL;//Minimales Regelsignal
	f_Max:REAL;//Maximales Regelsignal
	f_Manuell:REAL;//Manuelles Regelsignal
	f_PFaktor:REAL;//Proportionalfaktor
	t_Takt:timestruct;//Regelungstakt
END_VAR
VAR_OUTPUT
	f_Regelsignal:REAL;//Regelsignal
END_VAR
VAR
END_VAR

IF x_Enable THEN//Wenn Ein wird berechnet	
	IF x_Manuell THEN//Wenn Manuell wird der Manuelle Wert auf den Ausgang geschrieben
		f_Regelsignal:=LIMIT(f_Min,f_Manuell,f_Max);
	ELSE//Sonst wird die Berechnung durchgeführt
		IF x_Invertiert THEN//Formel für Berechnung (Istwert - Sollwert - Offset) x P Faktor 
			f_Regelsignal:=LIMIT(f_Min,
							(f_Ist-f_Sollwert-f_Offset)*f_PFaktor,
							f_Max);
		ELSE//(Sollwert + Ossfet - Istwert) x P Faktor 
			f_Regelsignal:=LIMIT(f_Min,
							(f_Sollwert+f_Offset-f_Ist)*f_PFaktor,
							f_Max);
		END_IF
		
	END_IF
ELSE//Sonst wird Regelsignal auf 0 geschrieben
	f_Regelsignal:=0.0;
END_IF

END_FUNCTION_BLOCK

// Regler/PIRegler
(*Der PI Regler rechnet die Differenz zwischen dem Sollwert und dem Istwert aus und multipliziert diese mit dem P Faktor. 
Zudem rechnet er bei jedem Takt den I Anteil aus und addiert diesen auf mit dem P Anteil. Je grösser die Faktoren sind, desto schneller und instabiler wirde der Regler.
P Anteil:
Formel Normal: (Sollwert + Ossfet - Istwert) x P Faktor 
Formel Invertiert: (Istwert - Sollwert - Offset) x P Faktor 
I Anteil:
Formel: I Anteil + I Faktor x P Anteil
Regelsignal: P + I Anteil
*)
FUNCTION_BLOCK PIRegler
(*
Versionsverlauf: 
Version		|Autor	|Bemerkung
------------------------------------------------------------------------------------------------------------ 
17.06.00	|Shgb	|erste Freigabe 
17.06.01	|ShgB	|von Integer auf Real geändert	
17.06.02	|ShgB	|Von Time auf Timestruct geändert
17.07.00	|ShgB	|Offset und Invertierung geändert.	
17.08.00	|LeaF	|Freigabe

*)
VAR_INPUT
	x_Enable:BOOL;//Freigabe des Reglers
	f_Ist:REAL;//Istwert
END_VAR
VAR_INPUT PERSISTENT
	x_Invertiert:BOOL;//Bei Kühlfunktionen aktiv
	x_Manuell:BOOL;//Manuelles Regelsignal aktivieren
	f_Sollwert:REAL;//Sollwertvorgabe
	f_Offset:REAL;//Offset
	f_Min:REAL;//Minimales Regelsignal
	f_Max:REAL;//Maximales Regelsignal
	f_Manuell:REAL;//Manuelles Regelsignal
	f_PFaktor:REAL;//Proportionalfaktor
	f_IFaktor:REAL;//Integralfaktor
	t_Takt:timestruct;//Regelungstakt
END_VAR
VAR_OUTPUT
	f_Regelsignal:REAL;//Regelsignal
END_VAR
VAR
	f_IAnteil,f_ISpeicher:REAL;
	f_PAnteil:REAL;
	P_Anteil: PRegler;
	Timer: TON;
	x_Takt:BOOL;
	Timestruct_to_Time:Timestruct_to_Time;
END_VAR

//P Anteil	
	P_Anteil(
		x_Enable:= x_Enable, 
		x_Invertiert:= x_Invertiert, 
		x_Manuell:= FALSE, 
		f_Sollwert:= f_Sollwert, 
		f_Ist:= f_Ist, 
		f_Offset:= f_Offset, 
		f_Min:= -f_Max, 
		f_Max:= f_Max, 
		f_Manuell:= 0, 
		f_PFaktor:= f_PFaktor, 
		f_Regelsignal=> f_PAnteil);

//TImestruct to Time
	Timestruct_to_Time(t_Ein:=t_Takt);
	
//Takt
	Timer(IN:= x_Enable AND NOT x_Takt, PT:= Timestruct_to_Time.t_Aus, Q=> x_Takt, ET=> );
	
//I Anteil
	IF x_Takt AND f_Regelsignal<f_Max AND f_Regelsignal>f_Min THEN
		f_ISpeicher:=f_ISpeicher+f_IFaktor*f_PAnteil;
	END_IF

//Reset Speicher
	IF NOT x_Enable THEN
		f_ISpeicher:=0.0;
	END_IF
	
//Grenzen einhalten	
	f_Regelsignal := LIMIT(f_Min,f_ISpeicher+f_PAnteil,f_Max);
	
//Manuell	
	IF x_Manuell THEN
		f_Regelsignal:=f_Manuell;
	END_IF

END_FUNCTION_BLOCK

// Timer/BLINK_A
(*Wenn x_Ein auf true blinkt der digitale Ausgang in einem asymetrischen Takt, mit den eingegebenen t_BlinkEin und t_BlinkAus Zeiten.
*)
FUNCTION_BLOCK BLINK_A
(*
Versionsverlauf: 
Version		|Autor	|Bemerkung
------------------------------------------------------------------------------------------------------------ 
17.05.00	|KuzR	|erste Freigabe 
17.08.00	|LeaF	|Freigabe

*)
VAR_INPUT
	x_Ein:BOOL;//Eingang Start
END_VAR
VAR_INPUT PERSISTENT
	t_BlinkEin:Timestruct := (wSecond := 5);//Zeiteingabe blinken Ein
	t_BlinkAus:Timestruct := (wSecond := 1);//Zeiteingabe blinken Aus
END_VAR
VAR_OUTPUT
	x_Aus:BOOL;//Digitaler Ausgang
END_VAR
VAR
	Blink:tof;		
	Pause:tof;
	t_PtZeitEIN:TIME;
	t_PtZeitAUS:TIME;
	Timestruct_to_Time: Timestruct_to_Time;
END_VAR

//Wenn Eingang True, dann läuft eingestellte Zeit ab, Ausgang True
	Timestruct_to_Time(t_Ein:=t_BlinkEin , t_Aus=>t_PtZeitEIN );
	Blink(in:=x_Ein AND NOT Pause.Q AND NOT Blink.Q, pt:=t_PtZeitEIN, Q=> x_Aus);

//Pause, läuft eingestellte Zeit ab, Ausgang False
	Timestruct_to_Time(t_Ein:=t_BlinkAus , t_Aus=>t_PtZeitAUS );
	Pause(in:=NOT Pause.Q AND NOT blink.Q, pt:=t_PtZeitAUS);

END_FUNCTION_BLOCK

// Timer/BLINK_S
(*Wenn x_Ein auf true blinkt der digitale Ausgang in einem symetrischen Takt, mit der eingegebenen t_BlinkEin Zeit.
*)
FUNCTION_BLOCK BLINK_S
(*
Versionsverlauf: 
Version		|Autor	|Bemerkung
------------------------------------------------------------------------------------------------------------ 
17.05.00	|KuzR	|erste Freigabe 
17.08.00	|LeaF	|Freigabe

*)
VAR_INPUT
	x_Ein:BOOL;
END_VAR
VAR_INPUT PERSISTENT
	t_BlinkEin:Timestruct := (wSecond := 5);
END_VAR
VAR_OUTPUT
	x_Aus:BOOL;
END_VAR
VAR
	Blink:tof;		
	Pause:tof;
	t_PtZeitEIN:TIME;
	Timestruct_to_Time:Timestruct_to_Time;	
END_VAR

//Wenn Eingang True, dann läuft eingestellte Zeit ab, Ausgang True
	Timestruct_to_Time(t_Ein:=t_BlinkEin, t_Aus=>t_PtZeitEIN );
	Blink(in:=x_Ein AND NOT Pause.Q AND NOT Blink.Q, pt:=t_PtZeitEIN, Q=> x_Aus);

//Pause, Ausgang False
	Timestruct_to_Time(t_Ein:=t_BlinkEin , t_Aus=>t_PtZeitEIN );
	Pause(in:=NOT Pause.Q AND NOT blink.Q, pt:=t_PtZeitEIN);

END_FUNCTION_BLOCK

// Timer/PULSE
(*Ist x_Ein auf true, wird x_Aus auf true gesetzt mit der eingegebenen Ablaufzeit. Sobald x_Ein auf false, dann x_Aus sofort auf false.
*)
FUNCTION_BLOCK PULSE
(*
Versionsverlauf: 
Version		|Autor	|Bemerkung
------------------------------------------------------------------------------------------------------------ 
17.05.00	|KuzR	|erste Freigabe 
17.08.00	|LeaF	|Freigabe

*)
VAR_INPUT
	x_Ein:BOOL;
END_VAR
VAR_INPUT PERSISTENT
	t_Abl:Timestruct := (wSecond := 5);//Eingegebene Ablaufzeit	
END_VAR
VAR_OUTPUT
	x_Aus:BOOL;//Digitaler Ausgang
	t_ET:Timestruct;//Ausgang Ablaufzeit
END_VAR
VAR
	Pulse:tp;
	t_PtZeit:TIME;
	Timestruct_to_Time:Timestruct_to_Time;	
	Time_to_Timestruct: Time_to_Timestruct;
END_VAR

//Wenn Eingang True, dann läuft eingestellte Zeit ab
	Timestruct_to_Time(t_Ein:=t_Abl , t_Aus=>t_PtZeit );
	Pulse(in:=x_Ein, pt:=t_PtZeit,Q=> x_Aus);

//Wenn Eingang False, dann Ausgang sofort auf False
	IF NOT x_Ein THEN
		x_Aus := FALSE;
	END_IF

//Ausgabe Ablaufzeit im timestruct
	Time_to_Timestruct(t_Ein:= Pulse.ET, t_Aus=> t_ET);

END_FUNCTION_BLOCK

// Timer/TOF_Reset
(*TOF Timer der mit einer Reset Funktion erweitert ist.
*)
FUNCTION_BLOCK TOF_Reset
(*
Versionsverlauf: 
Version		|Autor	|Bemerkung
------------------------------------------------------------------------------------------------------------ 
17.06.00	|Shgb	|erste Freigabe 
17.06.01	|ShgB	|Von Time auf Timestruct geändert
17.08.00	|LeaF	|Freigabe

*)
VAR_INPUT
	x_Ein:BOOL;//Eingang
	x_Reset:BOOL;//Ausschaltverzögerung wird auf 0 gesetzt
END_VAR
VAR_INPUT PERSISTENT
	t_time:timestruct := (wMinute := 5);//Ausschaltverzögerung
END_VAR
VAR_OUTPUT
	x_Aus:BOOL;//Ausgang
	t_Restzeit:timestruct;//Restzeit der Timerfunktion
END_VAR
VAR
	Timer: TOF;
	x_ResetFunktion:BOOL;
	Time_to_Timestruct: Time_to_Timestruct;
	Timestruct_to_Time:Timestruct_to_Time;
END_VAR

//Reset
	IF x_Reset THEN
		x_ResetFunktion := TRUE;
	END_IF

	IF x_Ein THEN
		x_ResetFunktion := FALSE;
	END_IF
	
//TImestruct to Time
	Timestruct_to_Time(t_Ein:=t_time);
	
//Beim Ausschalten Timer aktivieren	
	Timer(IN:=x_Ein, PT:= Timestruct_to_Time.t_Aus);

//Restzeit berechnen
	IF NOT x_ResetFunktion THEN
		Time_to_Timestruct(t_Ein:= Timestruct_to_Time.t_Aus-timer.ET, t_Aus=> t_Restzeit);
	ELSE
		Time_to_Timestruct(t_Ein:= T#0S, t_Aus=> t_Restzeit);
	END_IF
	
//Ausgang schalten
	x_Aus:=timer.Q AND NOT x_ResetFunktion;

END_FUNCTION_BLOCK

// Timer/TON_Reset
(*TON Timer der mit einer Reset Funktion erweitert ist.
*)
FUNCTION_BLOCK TON_Reset
(*
Versionsverlauf: 
Version		|Autor	|Bemerkung
------------------------------------------------------------------------------------------------------------ 
17.06.00	|Shgb	|erste Freigabe 
17.08.00	|LeaF	|Freigabe

*)
VAR_INPUT
	x_Ein:BOOL;//Eingang
	x_Reset:BOOL;//Einschaltverzögerung wird auf 0 gesetzt
END_VAR
VAR_INPUT PERSISTENT
	t_time:timestruct := (wMinute := 5);//Ausschaltverzögerung
END_VAR
VAR_OUTPUT
	x_Aus:BOOL;//Ausgang
	t_Restzeit:timestruct;//Restzeit der Timerfunktion
END_VAR
VAR
	Timer: TON;
	x_Timer,x_ResetFunktion:BOOL;
	t_ET:TIME;
	Time_to_Timestruct: Time_to_Timestruct;
	Timestruct_to_Time:Timestruct_to_Time;
END_VAR

//Reset
	IF x_Reset THEN
		x_ResetFunktion := TRUE;
	END_IF

	IF NOT x_Ein THEN
		x_ResetFunktion := FALSE;
	END_IF
	
//TImestruct to Time
	Timestruct_to_Time(t_Ein:=t_time);
	
//Beim Einschalten Timer aktivieren	
	Timer(IN:= x_Ein, PT:= Timestruct_to_Time.t_Aus, Q=> x_timer, ET=> t_ET);

//Restzeit berechnen
	IF NOT x_ResetFunktion THEN
		Time_to_Timestruct(t_Ein:= Timestruct_to_Time.t_Aus-t_ET, t_Aus=> t_Restzeit);
	ELSE
		Time_to_Timestruct(t_Ein:= T#0S, t_Aus=> t_Restzeit);
	END_IF
	
//Ausgang schalten
	x_Aus:= x_timer OR x_ResetFunktion;

END_FUNCTION_BLOCK

// Timer/Work
(*Betriebstunden- und Impulszäheler
*)
FUNCTION_BLOCK Work
(*
Versionsverlauf: 
Version		|Autor	|Bemerkung
------------------------------------------------------------------------------------------------------------ 
17.06.00	|Shgb	|erste Freigabe 
17.08.00	|ShgB	|Betriebsstunden nicht mit DT berechnet da Time Format nur bis 49 Tage geht.

*)
VAR_INPUT
	x_Ein:BOOL;//Eingang
	x_Reset:BOOL;//Stellt die Zähler auf 0 zurück
END_VAR
VAR_INPUT PERSISTENT
	t_StartBetriebsstunden:TIMESTRUCT;//Betriebsstunden die bei einem Reset auf den Ausgang geschrieben werden
	i_StartEinschaltungen:INT;//Anzahl Einschaltungen die bei einem Reset auf den Ausgang geschriben werden
END_VAR
VAR_OUTPUT PERSISTENT
	t_Betriebsstunden:TIMESTRUCT;//Anzeige der bis jetzt geleisteten Betriebsstunden
	i_Einschaltungen:INT;//Anzeige Einschaltimpulse
END_VAR
VAR
	x_Speicher: BOOL;
	w_Speicher:WORD;
END_VAR

//Impulse zählen
	IF x_Ein AND NOT x_Speicher THEN
		i_Einschaltungen:= i_Einschaltungen+1;
	END_IF
	x_Speicher:=x_Ein;
	
//Betriebsstundenzähler
	IF x_Ein THEN
		IF w_Speicher <> Globale_Uhr.systemtimestruct.wSecond THEN
			t_Betriebsstunden.wSecond := t_Betriebsstunden.wSecond +1;
			IF t_Betriebsstunden.wSecond>=60 THEN
				t_Betriebsstunden.wSecond:=0;
				t_Betriebsstunden.wMinute:=t_Betriebsstunden.wMinute+1;
				IF t_Betriebsstunden.wMinute>=60 THEN
					t_Betriebsstunden.wMinute:=0;
					t_Betriebsstunden.wHour:=t_Betriebsstunden.wHour+1;
					IF t_Betriebsstunden.wHour >=24 THEN
						t_Betriebsstunden.wHour:=0;
						t_Betriebsstunden.wDay:=t_Betriebsstunden.wDay+1;						
					END_IF
				END_IF
			END_IF
			w_Speicher:=Globale_Uhr.systemtimestruct.wSecond;
		END_IF
	END_IF	

//Reset
	IF x_Reset THEN
		i_Einschaltungen:=i_StartEinschaltungen;
		t_Betriebsstunden:=t_StartBetriebsstunden;
	END_IF

END_FUNCTION_BLOCK

// Timer/XPULSE
(*Ist x_Ein auf true, wird x_Aus auf true gesetzt mit der eingegebenen Ablaufzeit, unabhängig ob x_Ein früher abfällt,
als die eingegebene Ablaufzeit.
*)
FUNCTION_BLOCK XPULSE
(*
Versionsverlauf: 
Version		|Autor	|Bemerkung
------------------------------------------------------------------------------------------------------------ 
17.05.00	|KuzR	|erste Freigabe 
17.08.00	|LeaF	|Freigabe

*)
VAR_INPUT
	x_Ein:BOOL;//Eingang
END_VAR
VAR_INPUT PERSISTENT
	t_Abl:Timestruct := (wSecond := 5);//Eingegebene Ablaufzeit	
END_VAR
VAR_OUTPUT
	x_Aus:BOOL;//Digitaler Ausgang
	t_ET:Timestruct;//Ausgang Ablaufzeit
END_VAR	
VAR
	Ein:tp;
	t_PtZeit:TIME;
	Timestruct_to_Time:Timestruct_to_Time;
	Time_to_Timestruct: Time_to_Timestruct;	
END_VAR

//Wenn Eingang True, dann läuft eingestellte Zeit ab	
	Timestruct_to_Time(t_Ein:=t_Abl , t_Aus=>t_PtZeit );
	Ein(IN:= x_Ein, PT:= t_PtZeit, Q=> x_Aus);

//Ausgabe Ablaufzeit im timestruct
	Time_to_Timestruct(t_Ein:= Ein.ET, t_Aus=> t_ET);

END_FUNCTION_BLOCK

// Uhren/ABS_Bool
(*Anti Blockiersystem für BOOL Aktoren. Wird der Aktor während der eingestellten Zeit nicht bewegt so wird dieser für eine bestimmte Dauer eingeschalten.
*)
FUNCTION_BLOCK ABS_Bool
(*
Versionsverlauf: 
Version		|Autor	|Bemerkung
------------------------------------------------------------------------------------------------------------ 
17.06.00	|Shgb	|erste Freigabe 

*)
VAR_INPUT
	x_Ein:BOOL;//Eingang
END_VAR
VAR_INPUT PERSISTENT
	t_Einschaltzeitpunkt:timestruct := (wDayOfWeek := 1, wHour := 9) ;//Wochentag mit Uhrzeit wann der Ausgang geschalten wird
	t_Dauer:timestruct := (wMinute := 2);//Dauer des Force Zycklus
END_VAR
VAR_OUTPUT
	x_Aus:BOOL;//Ausgang
END_VAR
VAR
	TOF:TOF;
	Dauer:Timestruct_to_Time;
	x_Bewegt: BOOL;
	x_Flanke: BOOL;
END_VAR

// Einschalten jede Woche, eingestellte Zeit
	IF  Globale_Uhr.systemtimestruct.wDayOfWeek = t_Einschaltzeitpunkt.wDayOfWeek  AND
		Globale_Uhr.systemtimestruct.wHour = t_Einschaltzeitpunkt.wHour AND
		Globale_Uhr.systemtimestruct.wMinute = t_Einschaltzeitpunkt.wMinute THEN
		IF NOT x_Bewegt AND NOT x_Flanke THEN
			TOF.IN:=TRUE;
		ELSE
			x_Bewegt:=FALSE;
		END_IF
		x_Flanke:=TRUE;
	ELSE
		x_Flanke:=FALSE;
	END_IF
	
//Sobald Bewegt wurde Bit setzen
	IF x_Ein THEN
		x_Bewegt:=TRUE;
	END_IF

//Timestruct to Time
	Dauer(t_Ein:=t_Dauer);
	TOF(PT:=Dauer.t_Aus);
	TOF.IN:=FALSE;

//Ausgang setzen
	x_Aus:=x_Ein OR tof.Q;

END_FUNCTION_BLOCK

// Uhren/ABS_Int
(*Anti Blockiersystem für INT Aktoren. Der Aktor wir nach Ablauf der eingestellten Zeit auf den i_Force Wert bewegt und bleibt währen der Dauer auf diesem Wert.
*)
FUNCTION_BLOCK ABS_Int
(*
Versionsverlauf: 
Version		|Autor	|Bemerkung
------------------------------------------------------------------------------------------------------------ 
17.06.00	|Shgb	|erste Freigabe 

*)
VAR_INPUT
	i_Ein:int;//Eingang
END_VAR
VAR_INPUT PERSISTENT 
	t_Einschaltzeitpunkt:timestruct := (wDay := 7);//Zeit zwischen den einzelnen Force Zycklen
	t_Dauer:timestruct := (wMinute := 2);//Dauer des Force Zycklus
END_VAR
VAR_OUTPUT
	i_Aus:INT;//Ausgang
END_VAR
VAR
	TOF: TOF;
	Dauer: Timestruct_to_Time;
	x_Bewegt: BOOL;
	i_Speicher: INT;
	x_Flanke: BOOL;
END_VAR

// Einschalten jede Woche, eingestellte Zeit
	IF  Globale_Uhr.systemtimestruct.wDayOfWeek = t_Einschaltzeitpunkt.wDayOfWeek  AND
		Globale_Uhr.systemtimestruct.wHour = t_Einschaltzeitpunkt.wHour AND
		Globale_Uhr.systemtimestruct.wMinute = t_Einschaltzeitpunkt.wMinute THEN
		IF NOT x_Bewegt AND NOT x_Flanke THEN
			TOF.IN:=TRUE;
		ELSE
			x_Bewegt:=FALSE;
			i_Speicher:=i_Ein;
		END_IF
		x_Flanke:=TRUE;
	ELSE
		x_Flanke:=FALSE;
	END_IF
	
//Sobald Bewegt wurde Bit setzen
	IF i_Ein >= i_Speicher+10 OR i_Ein <= i_Speicher-10 THEN
		x_Bewegt:=TRUE;
	END_IF

//Timestruct to Time
	Dauer(t_Ein:=t_Dauer);
	TOF(PT:=Dauer.t_Aus);
	TOF.IN:=FALSE;

//Ausgang setzen
	IF tof.Q THEN
		i_Aus:=1000-i_Ein;	
	ELSE
		i_Aus:=i_Ein;
	END_IF;

END_FUNCTION_BLOCK

// Uhren/ABS_Real
(*Anti Blockiersystem für REAL Aktoren. Der Aktor wir nach Ablauf der eingestellten Zeit auf den f_Force Wert bewegt und bleibt währen der Dauer auf diesem Wert.
*)
FUNCTION_BLOCK ABS_Real
(*
Versionsverlauf: 
Version		|Autor	|Bemerkung
------------------------------------------------------------------------------------------------------------ 
17.06.00	|Shgb	|erste Freigabe 

*)
VAR_INPUT
	f_Ein:real;//Eingang
END_VAR
VAR_INPUT PERSISTENT 
	t_Einschaltzeitpunkt:timestruct := (wDay := 7);//Zeit zwischen den einzelnen Force Zycklen
	t_Dauer:timestruct := (wMinute := 2);//Dauer des Force Zycklus
END_VAR
VAR_OUTPUT
	f_Aus:REAL;//Ausgang
END_VAR
VAR
	TOF: TOF;
	Dauer: Timestruct_to_Time;
	x_Bewegt: BOOL;
	f_Speicher: REAL;

	x_Flanke: BOOL;
END_VAR

// Einschalten jede Woche, eingestellte Zeit
	IF  Globale_Uhr.systemtimestruct.wDayOfWeek = t_Einschaltzeitpunkt.wDayOfWeek  AND
		Globale_Uhr.systemtimestruct.wHour = t_Einschaltzeitpunkt.wHour AND
		Globale_Uhr.systemtimestruct.wMinute = t_Einschaltzeitpunkt.wMinute THEN
		IF NOT x_Bewegt AND NOT x_Flanke THEN
			TOF.IN:=TRUE;
		ELSE
			x_Bewegt:=FALSE;
			f_Speicher:=f_Ein;
		END_IF
		x_Flanke:=TRUE;
	ELSE
		x_Flanke:=FALSE;
	END_IF
	
//Sobald Bewegt wurde Bit setzen
	IF f_Ein >= f_Speicher+10 OR f_Ein <= f_Speicher-10 THEN
		x_Bewegt:=TRUE;
	END_IF

//Timestruct to Time
	Dauer(t_Ein:=t_Dauer);
	TOF(PT:=Dauer.t_Aus);
	TOF.IN:=FALSE;

//Ausgang setzen
	IF tof.Q THEN
		f_Aus:=100-f_Ein;	
	ELSE
		f_Aus:=f_Ein;
	END_IF;

END_FUNCTION_BLOCK

// Uhren/CLK_I
(*Uhr mit einem Impuls pro Tag. Einschaltzeit => t_Ein.wHour, t_ein.wMinute und Impulszeit => t_Imp.w.Second Eingabe im Timestruct Format. Vergleicht Einschaltzeit 
mit der Globalen_Uhr(Globale Variable)
*)
FUNCTION_BLOCK CLK_I
(*
Versionsverlauf: 
Version		|Autor	|Bemerkung
------------------------------------------------------------------------------------------------------------ 
17.06.00	|KuzR	|erste Freigabe 
17.08.00	|LeaF	|Freigabe

*)
VAR_INPUT Persistent
 	t_Ein:timestruct;//Eingabe Einschaltzeit 
	t_Imp:timestruct;//Eingabe Impulszeit
END_VAR
VAR_OUTPUT
	x_Aus:BOOL;//Digitaler Ausgang			 
END_VAR
VAR	
	impuls:tp;
	x_Zeit_groesser:BOOL;   
	t_ptImpuls: TIME;
	Timestruct_to_Time: Timestruct_to_Time;
END_VAR

//schaltet jeden Tag ein, eingestellte Zeit
	IF Globale_Uhr.systemtimestruct.wHour = t_Ein.wHour AND
 	   Globale_Uhr.systemtimestruct.wMinute >= t_Ein.wMinute THEN
			x_Zeit_groesser	:=TRUE;		
	ELSE
			x_Zeit_groesser :=  FALSE;
	END_IF
				
//Impulsdauer
	Timestruct_to_Time(t_Ein:=t_Imp , t_Aus=>t_ptImpuls );
	impuls(in:=x_Zeit_groesser, pt:=t_ptImpuls);
		x_Aus:= impuls.Q;
		x_Zeit_groesser:= x_Aus;

END_FUNCTION_BLOCK

// Uhren/CLK_M
(*Uhr mit Monatsprogramm. Schaltet 1mal im Monat für eine einstellbare Zeit.  Einschaltzeit => t_Ein.wDay, t_Ein.wHour, t_ein.wMinute
und Ausschaltzeit => t_Ein.wDay, t_Ein.wHour, t_ein.wMinute.
Eingabe im Timestruct Format. Vergleicht Ein- und Ausschaltzeit mit der Globalen_Uhr(Globale Variable)
*)
FUNCTION_BLOCK CLK_M
(*
Versionsverlauf: 
Version		|Autor	|Bemerkung
------------------------------------------------------------------------------------------------------------ 
17.06.00	|KuzR	|erste Freigabe 
17.08.00	|LeaF	|Freigabe

*)
VAR_INPUT Persistent
	    t_Ein:timestruct;//Eingabe Einschaltzeit 
		t_Aus:timestruct;//Eingabe Ausschaltzeit 	
END_VAR
VAR_OUTPUT
		x_Aus:BOOL;	 
END_VAR
VAR
	
		
	
	
	

		
	
	
END_VAR

// Einschalten einmal im Monat, Tag und Zeit
	IF  Globale_Uhr.systemtimestruct.wDay = t_Ein.wDay  AND
		Globale_Uhr.systemtimestruct.wHour = t_Ein.wHour AND
		Globale_Uhr.systemtimestruct.wMinute >= t_Ein.wMinute THEN
			x_Aus:= TRUE;
	END_IF
	
// Ausschalten einmal im Monat, Tag und Zeit
	IF  Globale_Uhr.systemtimestruct.wDay = t_Aus.wDay  AND
		Globale_Uhr.systemtimestruct.wHour = t_Aus.wHour AND
		Globale_Uhr.systemtimestruct.wMinute >= t_Aus.wMinute THEN
			x_Aus:= FALSE;
	END_IF

END_FUNCTION_BLOCK

// Uhren/CLK_W
(*Uhr mit Wochernprogramm. Schaltet 1 mal in der Woche für eine einstellbare Zeit.  Einschaltzeit => t_Ein.wDayofWeek, t_Ein.wHour, t_ein.wMinute
und Ausschaltzeit => t_Ein.wDayofWeek, t_Ein.wHour, t_ein.wMinute.
Eingabe im Timestruct Format. Vergleicht Ein- und Ausschaltzeit mit der Globalen_Uhr(Globale Variable)
*)
FUNCTION_BLOCK CLK_W
(*
Versionsverlauf: 
Version		|Autor	|Bemerkung
------------------------------------------------------------------------------------------------------------ 
17.06.00	|KuzR	|erste Freigabe 
17.08.00	|LeaF	|Freigabe

*)
VAR_INPUT Persistent
	t_Ein:timestruct;//Eingabe Einschaltzeit 
	t_Aus:timestruct;//Eingabe Ausschaltzeit
END_VAR
VAR_OUTPUT
	x_Aus:BOOL;//Digitaler Ausgang 
END_VAR

// Einschalten jede Woche, eingestellte Zeit
	IF  Globale_Uhr.systemtimestruct.wDayOfWeek = t_Ein.wDayOfWeek  AND
		Globale_Uhr.systemtimestruct.wHour = t_Ein.wHour AND
		Globale_Uhr.systemtimestruct.wMinute >= t_Ein.wMinute THEN
			x_Aus:= TRUE;
	END_IF
// Ausschalten, eingestellte Zeit
	IF  Globale_Uhr.systemtimestruct.wDayOfWeek = t_Aus.wDayOfWeek  AND
		Globale_Uhr.systemtimestruct.wHour = t_Aus.wHour AND
		Globale_Uhr.systemtimestruct.wMinute >= t_Aus.wMinute THEN
			x_Aus:= FALSE;
	END_IF

END_FUNCTION_BLOCK

// Uhren/CLK_W7
(*Uhr mit Wochenprogramm für jeden Wochentag. Schaltet 1 mal im Tag für eine einstellbare Zeit, jeden Wochentag einzeln wählbar.
Einschaltzeit => t_Ein.wHour, t_ein.wMinute
und Ausschaltzeit => t_Ein.wHour, t_ein.wMinute
Eingabe im Timestruct Format. Vergleicht Ein- und Ausschaltzeit mit der Globalen_Uhr(Globale Variable)
*)
FUNCTION_BLOCK CLK_W7
(*
Versionsverlauf: 
Version		|Autor	|Bemerkung
------------------------------------------------------------------------------------------------------------ 
17.06.00	|KuzR	|erste Freigabe 
17.08.00	|LeaF	|Freigabe

*)
VAR_INPUT Persistent	   	
		t_Ein_Mo:timestruct;//Eingabe Einschaltzeit Montag
		t_Aus_Mo:timestruct;//Eingabe Ausschaltzeit Montag
 		t_Ein_Di:timestruct;//Eingabe Einschaltzeit Dienstag
		t_Aus_Di:timestruct;//Eingabe Ausschaltzeit Dienstag
		t_Ein_Mi:timestruct;//Eingabe Einschaltzeit Mittwoch
		t_Aus_Mi:timestruct;//Eingabe Ausschaltzeit Mittwoch
		t_Ein_Do:timestruct;//Eingabe Einschaltzeit Donnerstag
		t_Aus_Do:timestruct;//Eingabe Ausschaltzeit Donnerstag
		t_Ein_Fr:timestruct;//Eingabe Einschaltzeit Freitag
		t_Aus_Fr:timestruct;//Eingabe Ausschaltzeit Freitag
		t_Ein_Sa:timestruct;//Eingabe Einschaltzeit Samstag
		t_Aus_Sa:timestruct;//Eingabe Ausschaltzeit Samstag
		t_Ein_So:timestruct;//Eingabe Einschaltzeit Sonntag
		t_Aus_So:timestruct;//Eingabe Ausschaltzeit Sonntag
END_VAR
VAR_OUTPUT
		x_Aus:BOOL;//Digitaler Ausgang	 
END_VAR
VAR
END_VAR

//Montag einschalten
	IF  Globale_Uhr.systemtimestruct.wDayOfWeek = 1  AND
		Globale_Uhr.systemtimestruct.wHour = t_Ein_Mo.wHour AND
		Globale_Uhr.systemtimestruct.wMinute >= t_Ein_Mo.wMinute THEN
			x_Aus:= TRUE;
			END_IF
//Montag ausschalten	
	IF  Globale_Uhr.systemtimestruct.wDayOfWeek = 1  AND
		Globale_Uhr.systemtimestruct.wHour = t_Aus_MO.wHour AND
		Globale_Uhr.systemtimestruct.wMinute >= t_Aus_MO.wMinute THEN
			x_Aus:= FALSE;
			END_IF
//Dienstag einschalten
	IF  Globale_Uhr.systemtimestruct.wDayOfWeek = 2  AND
		Globale_Uhr.systemtimestruct.wHour = t_Ein_Di.wHour AND
		Globale_Uhr.systemtimestruct.wMinute >= t_Ein_Di.wMinute THEN
			x_Aus:= TRUE;
			END_IF
//Dienstag ausschalten	
	IF  Globale_Uhr.systemtimestruct.wDayOfWeek = 2  AND
		Globale_Uhr.systemtimestruct.wHour = t_Aus_Di.wHour AND
		Globale_Uhr.systemtimestruct.wMinute >= t_Aus_Di.wMinute THEN
			x_Aus:= FALSE;
			END_IF
//Mittwoch einschalten
	IF  Globale_Uhr.systemtimestruct.wDayOfWeek = 3  AND
		Globale_Uhr.systemtimestruct.wHour = t_Ein_Mi.wHour AND
		Globale_Uhr.systemtimestruct.wMinute >= t_Ein_Mi.wMinute THEN
			x_Aus:= TRUE;
			END_IF
//Mittwoch ausschalten	
	IF  Globale_Uhr.systemtimestruct.wDayOfWeek = 3  AND
		Globale_Uhr.systemtimestruct.wHour = t_Aus_Mi.wHour AND
		Globale_Uhr.systemtimestruct.wMinute >= t_Aus_Mi.wMinute THEN
			x_Aus:= FALSE;
			END_IF		
//Donnerstag einschalten
	IF  Globale_Uhr.systemtimestruct.wDayOfWeek = 4  AND
		Globale_Uhr.systemtimestruct.wHour = t_Ein_Do.wHour AND
		Globale_Uhr.systemtimestruct.wMinute >= t_Ein_Do.wMinute THEN
			x_Aus:= TRUE;
			END_IF
//Donnerstag ausschalten	
	IF  Globale_Uhr.systemtimestruct.wDayOfWeek = 4  AND
		Globale_Uhr.systemtimestruct.wHour = t_Aus_Do.wHour AND
		Globale_Uhr.systemtimestruct.wMinute >= t_Aus_Do.wMinute THEN
			x_Aus:= FALSE;
			END_IF

//Freitag einschalten
	IF  Globale_Uhr.systemtimestruct.wDayOfWeek = 5  AND
		Globale_Uhr.systemtimestruct.wHour = t_Ein_Fr.wHour AND
		Globale_Uhr.systemtimestruct.wMinute >= t_Ein_Fr.wMinute THEN
			x_Aus:= TRUE;
			END_IF
//Freitag ausschalten	
	IF  Globale_Uhr.systemtimestruct.wDayOfWeek = 5  AND
		Globale_Uhr.systemtimestruct.wHour = t_Aus_Fr.wHour AND
		Globale_Uhr.systemtimestruct.wMinute >= t_Aus_Fr.wMinute THEN
			x_Aus:= FALSE;
			END_IF		
//Samstag einschalten
	IF  Globale_Uhr.systemtimestruct.wDayOfWeek = 6  AND
		Globale_Uhr.systemtimestruct.wHour = t_Ein_Sa.wHour AND
		Globale_Uhr.systemtimestruct.wMinute >= t_Ein_Sa.wMinute THEN
			x_Aus:= TRUE;
			END_IF
//Samstag ausschalten	
	IF  Globale_Uhr.systemtimestruct.wDayOfWeek = 6  AND
		Globale_Uhr.systemtimestruct.wHour = t_Aus_Sa.wHour AND
		Globale_Uhr.systemtimestruct.wMinute >= t_Aus_Sa.wMinute THEN
			x_Aus:= FALSE;
			END_IF	
//Sonntag einschalten
	IF  Globale_Uhr.systemtimestruct.wDayOfWeek = 0  AND
		Globale_Uhr.systemtimestruct.wHour = t_Ein_So.wHour AND
		Globale_Uhr.systemtimestruct.wMinute >= t_Ein_So.wMinute THEN
			x_Aus:= TRUE;
			END_IF
//Sonntag ausschalten	
	IF  Globale_Uhr.systemtimestruct.wDayOfWeek = 0  AND
		Globale_Uhr.systemtimestruct.wHour = t_Aus_So.wHour AND
		Globale_Uhr.systemtimestruct.wMinute >= t_Aus_So.wMinute THEN
			x_Aus:= FALSE;
			END_IF

END_FUNCTION_BLOCK

// Uhren/CLK_Y
(*Uhr mit Jahresrogramm. Schaltet 1 mal im Jahr für eine einstellbare Zeit.  Einschaltzeit => t_Ein.wMonth, t_Ein.wDay, t_Ein.wHour, t_ein.wMinute
und Ausschaltzeit => t_Aus.wMonth, t_Ein.wDay, t_Ein.wHour, t_ein.wMinute.
Eingabe im Timestruct Format. Vergleicht Ein- und Ausschaltzeit mit der Globalen_Uhr(Globale Variable)
*)
FUNCTION_BLOCK CLK_Y
(*
Versionsverlauf: 
Version		|Autor	|Bemerkung
------------------------------------------------------------------------------------------------------------ 
17.06.00	|KuzR	|erste Freigabe 
17.08.00	|LeaF	|Freigabe

*)
VAR_INPUT Persistent
	t_Ein:timestruct;//Eingabe Einschaltzeit
	t_Aus:timestruct;//Eingabe Ausschaltzeit	

END_VAR
VAR_OUTPUT
	x_Aus:BOOL;			 
END_VAR
VAR
END_VAR

// Einschalten einmal im Jahr, Zeit, Tagnummer und Monat
	IF Globale_Uhr.systemtimestruct.wMonth = t_Ein.wMonth AND
 	   Globale_Uhr.systemtimestruct.wDay = t_Ein.wDay AND
	   Globale_Uhr.systemtimestruct.wHour = t_Ein.wHour AND
	   Globale_Uhr.systemtimestruct.wMinute >= t_Ein.wMinute THEN
			x_Aus:= TRUE;		
	END_IF
			
// Ausschalten Zeit, Tagnummer und Monat 	
	IF Globale_Uhr.systemtimestruct.wMonth = t_Aus.wMonth AND
 	   Globale_Uhr.systemtimestruct.wDay = t_Aus.wDay AND
	   Globale_Uhr.systemtimestruct.wHour = t_Aus.wHour AND
	   Globale_Uhr.systemtimestruct.wMinute >= t_Aus.wMinute THEN			
			x_Aus:= FALSE;
	END_IF

END_FUNCTION_BLOCK

// Uhren/FerienPRG
(*FB Ferienprogramm, Wenn FB aktiviert und die Schaltuhr aktiv ist, schaltet die Freigabe x_BM und der Sollwert Eingang wird auf
den Ausgang geschrieben. Es muss nur die Ausschaltzeit eingegeben werden t_Aus.wMonth, => t_Aus.wDay, t_Aus.wHour, t_Aus.wMinute.
Sobald die Zeit abgelaufen ist, wird der Sollwert Ausgang auf 0 gesetzt und der Ausgang x_BM wird auf false gesetzt.
*)
FUNCTION_BLOCK FerienPRG
(*
Versionsverlauf: 
Version		|Autor	|Bemerkung
------------------------------------------------------------------------------------------------------------ 
17.07.00	|KuzR	|erste Freigabe 
17.08.00	|LeaF	|Freigabe

*)
VAR_INPUT PERSISTENT
	x_Akt:BOOL;//Aktivierung
	t_Aus:TIMESTRUCT;//Ausschaltzeit
	f_SW_fix:REAL;//Sollwert
END_VAR
VAR_OUTPUT
	x_BM:BOOL;//Freigabe
	f_SW:REAL;//Sollwert
	t_Restzeit:timestruct;//Anzeige Restzeit
END_VAR
VAR
	ein: BOOL;
	x_Aus_Uhr:BOOL;
	x_ein:BOOL;
	t_Restzeit1:TIME;
	t_Ausschalt: TIME;
	t_Global:TIME;
	CLK_M: CLK_M;
	Timestruct_to_Time: Timestruct_to_Time;
	Time_to_Timestruct: Time_to_Timestruct;
	SWITCH_REAL: SWITCH_REAL;
	
	CLK_Y: CLK_Y;
END_VAR

//Kommentar

//Monatsuhr, Zeiteingabe im Timestruct
		CLK_Y(t_Ein:= Globale_Uhr.systemtimestruct, t_Aus:=t_Aus , x_Aus=>x_Aus_Uhr );
//Freigabe schalten
 		x_BM:= x_Akt AND x_Aus_Uhr;

//Timestruct to time
		Timestruct_to_Time(t_Ein:=t_Aus , t_Aus=>t_Ausschalt );
		Timestruct_to_Time(t_Ein:=Globale_Uhr.systemtimestruct , t_Aus=>t_Global);	
			
//Restzeit berechnen im Time Format
		t_Restzeit1:=t_Ausschalt-t_Global;
	IF t_Ausschalt < t_Global THEN
		t_Restzeit1:=T#0S;
	END_IF
	
//Time to timestruct
	Time_to_Timestruct(t_Ein:= t_Restzeit1, t_Aus=> t_Restzeit);

//Sollwert in den Ausgang schreiben	
	SWITCH_REAL(x_Ein:=x_BM , f_Ein_1:=0 , f_Ein_2:=f_SW_fix , f_Aus=>f_SW );
		
	IF NOT x_Aus_Uhr THEN
		x_Akt:=FALSE;
	END_IF

END_FUNCTION_BLOCK

// Verdichter/FIFO
(*Funktionsbaustein zum Abgleich der Betriebsstunden. Der Kompressor mit der geringeren Anzahl an Betriebsstunden wird als nächstes in Betrieb genommen. 
Beim Ausschalten werden die Kompressoren nach dem FIFO (First in frist out) Prinzip ausgeschalten.
*)
FUNCTION_BLOCK FIFO
(*
Versionsverlauf: 
Version		|Autor	|Bemerkung
------------------------------------------------------------------------------------------------------------ 
17.06.00	|Shgb	|erste Freigabe
17.07.00	|Shgb	|Bool zum Kompressorwechsel
17.08.00	|LeaF	|Freigabe

*)
VAR_INPUT
	i_Stufen:INT;//Anzahl der angeforderten Stufen
	x_En1:BOOL;//Betriebstunden von Kompressor 1
	t_Betriebsstunden1:timestruct;//Betriebstunden von Kompressor 1
	x_En2:BOOL;//Betriebstunden von Kompressor 2
	t_Betriebsstunden2:timestruct;//Betriebstunden von Kompressor 2
	x_En3:BOOL;//Betriebstunden von Kompressor 3
	t_Betriebsstunden3:timestruct;//Betriebstunden von Kompressor 3
	x_En4:BOOL;//Betriebstunden von Kompressor 4
	t_Betriebsstunden4:timestruct;//Betriebstunden von Kompressor 4
	x_En5:BOOL;//Betriebstunden von Kompressor 5
	t_Betriebsstunden5:timestruct;//Betriebstunden von Kompressor 5
	x_En6:BOOL;//Betriebstunden von Kompressor 6
	t_Betriebsstunden6:timestruct;//Betriebstunden von Kompressor 6
	x_En7:BOOL;//Betriebstunden von Kompressor 7
	t_Betriebsstunden7:timestruct;//Betriebstunden von Kompressor 7
	x_En8:BOOL;//Betriebstunden von Kompressor 8
	t_Betriebsstunden8:timestruct;//Betriebstunden von Kompressor 8
	x_Wechsel: BOOL;	// Befhel für die Umschaltung der betriebenen Kompressoren.
END_VAR
VAR_OUTPUT
	x_Aus1:BOOL;//Einschaltbefehl Kompressor 1
	x_Aus2:BOOL;//Einschaltbefehl Kompressor 2
	x_Aus3:BOOL;//Einschaltbefehl Kompressor 3
	x_Aus4:BOOL;//Einschaltbefehl Kompressor 4
	x_Aus5:BOOL;//Einschaltbefehl Kompressor 5
	x_Aus6:BOOL;//Einschaltbefehl Kompressor 6
	x_Aus7:BOOL;//Einschaltbefehl Kompressor 7
	x_Aus8:BOOL;//Einschaltbefehl Kompressor 8
END_VAR
VAR
	t_Ein1,t_Ein2,t_Ein3,t_Ein4:DT;
	t_Ein5,t_Ein6,t_Ein7,t_Ein8:DT;
	Count: COUNT;
	i_Count: INT;
	x_Speicher: BOOL;
	x_1_2: Timestruct_Kleiner_Gleich_Timestruct;
	x_1_3: Timestruct_Kleiner_Gleich_Timestruct;
	x_1_4: Timestruct_Kleiner_Gleich_Timestruct;
	x_1_5: Timestruct_Kleiner_Gleich_Timestruct;
	x_1_6: Timestruct_Kleiner_Gleich_Timestruct;
	x_1_7: Timestruct_Kleiner_Gleich_Timestruct;
	x_1_8: Timestruct_Kleiner_Gleich_Timestruct;
	x_2_1: Timestruct_Kleiner_Gleich_Timestruct;
	x_2_3: Timestruct_Kleiner_Gleich_Timestruct;
	x_2_4: Timestruct_Kleiner_Gleich_Timestruct;
	x_2_5: Timestruct_Kleiner_Gleich_Timestruct;
	x_2_6: Timestruct_Kleiner_Gleich_Timestruct;
	x_2_7: Timestruct_Kleiner_Gleich_Timestruct;
	x_2_8: Timestruct_Kleiner_Gleich_Timestruct;
	x_3_1: Timestruct_Kleiner_Gleich_Timestruct;
	x_3_2: Timestruct_Kleiner_Gleich_Timestruct;
	x_3_4: Timestruct_Kleiner_Gleich_Timestruct;
	x_3_5: Timestruct_Kleiner_Gleich_Timestruct;
	x_3_6: Timestruct_Kleiner_Gleich_Timestruct;
	x_3_7: Timestruct_Kleiner_Gleich_Timestruct;
	x_3_8: Timestruct_Kleiner_Gleich_Timestruct;
	x_4_1: Timestruct_Kleiner_Gleich_Timestruct;
	x_4_2: Timestruct_Kleiner_Gleich_Timestruct;
	x_4_3: Timestruct_Kleiner_Gleich_Timestruct;
	x_4_5: Timestruct_Kleiner_Gleich_Timestruct;
	x_4_6: Timestruct_Kleiner_Gleich_Timestruct;
	x_4_7: Timestruct_Kleiner_Gleich_Timestruct;
	x_4_8: Timestruct_Kleiner_Gleich_Timestruct;
	x_5_1: Timestruct_Kleiner_Gleich_Timestruct;
	x_5_2: Timestruct_Kleiner_Gleich_Timestruct;
	x_5_3: Timestruct_Kleiner_Gleich_Timestruct;
	x_5_4: Timestruct_Kleiner_Gleich_Timestruct;
	x_5_6: Timestruct_Kleiner_Gleich_Timestruct;
	x_5_7: Timestruct_Kleiner_Gleich_Timestruct;
	x_5_8: Timestruct_Kleiner_Gleich_Timestruct;
	x_6_1: Timestruct_Kleiner_Gleich_Timestruct;
	x_6_2: Timestruct_Kleiner_Gleich_Timestruct;
	x_6_3: Timestruct_Kleiner_Gleich_Timestruct;
	x_6_4: Timestruct_Kleiner_Gleich_Timestruct;
	x_6_5: Timestruct_Kleiner_Gleich_Timestruct;
	x_6_7: Timestruct_Kleiner_Gleich_Timestruct;
	x_6_8: Timestruct_Kleiner_Gleich_Timestruct;
	x_7_1: Timestruct_Kleiner_Gleich_Timestruct;
	x_7_2: Timestruct_Kleiner_Gleich_Timestruct;
	x_7_3: Timestruct_Kleiner_Gleich_Timestruct;
	x_7_4: Timestruct_Kleiner_Gleich_Timestruct;
	x_7_5: Timestruct_Kleiner_Gleich_Timestruct;
	x_7_6: Timestruct_Kleiner_Gleich_Timestruct;
	x_7_8: Timestruct_Kleiner_Gleich_Timestruct;
	x_8_1: Timestruct_Kleiner_Gleich_Timestruct;
	x_8_2: Timestruct_Kleiner_Gleich_Timestruct;
	x_8_3: Timestruct_Kleiner_Gleich_Timestruct;
	x_8_4: Timestruct_Kleiner_Gleich_Timestruct;
	x_8_5: Timestruct_Kleiner_Gleich_Timestruct;
	x_8_6: Timestruct_Kleiner_Gleich_Timestruct;
	x_8_7: Timestruct_Kleiner_Gleich_Timestruct;
END_VAR

